KUKA KRL program: MASTER_125_LADO_B.src, MASTER_125_LADO_B.dat

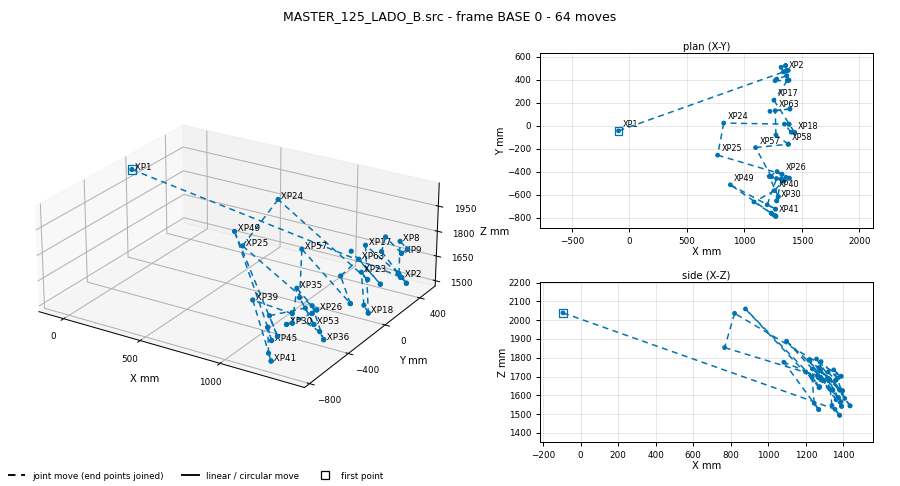
[picture p0: tool path of MASTER_125_LADO_B.src in frame BASE 0, 64 of 66 moves have a stored position in this frame; points joined in program order, loops and branches not executed]
--- MASTER_125_LADO_B.src ---
&ACCESS RVP
&REL 169
&PARAM EDITMASK = *
&PARAM TEMPLATE = C:\KRC\Roboter\Template\vorgabe
&PARAM DISKPATH = KRC:\R1\Program\Solda\MASTER_125
DEF MASTER_125_LADO_B( )
;FOLD INI;%{PE}
  ;FOLD BASISTECH INI
    GLOBAL INTERRUPT DECL 3 WHEN $STOPMESS==TRUE DO IR_STOPM ( )
    INTERRUPT ON 3
    BAS (#INITMOV,0 )
  ;ENDFOLD (BASISTECH INI)
  ;FOLD USER INI
    ;Make your modifications here

  ;ENDFOLD (USER INI)
;ENDFOLD (INI)
;FOLD OUT 128 'Perfil livre mesa B' State=FALSE CONT;%{PE}%R 8.3.48,%MKUKATPBASIS,%COUT,%VOUTX,%P 2:128, 3:Perfil livre mesa B, 5:FALSE, 6:CONTINUE
CONTINUE
$OUT[128]=FALSE
;ENDFOLD
;FOLD OUT 125 'Lado A para operador' State=TRUE ;%{PE}%R 8.3.48,%MKUKATPBASIS,%COUT,%VOUTX,%P 2:125, 3:Lado A para operador, 5:TRUE, 6:
$OUT[125]=TRUE
;ENDFOLD

;FOLD PTP HOME1 Vel=100 % PDAT2;%{PE}%R 8.3.48,%MKUKATPBASIS,%CMOVE,%VPTP,%P 1:PTP, 2:HOME1, 3:, 5:100, 7:PDAT2
$BWDSTART=FALSE
PDAT_ACT=PPDAT2
FDAT_ACT=FHOME1
BAS(#PTP_PARAMS,100)
PTP XHOME1
;ENDFOLD
;FOLD PTP P1 CONT Vel=100 % PDAT1 Tool[1]:TOCH Base[0];%{PE}%R 8.3.48,%MKUKATPBASIS,%CMOVE,%VPTP,%P 1:PTP, 2:P1, 3:C_DIS, 5:100, 7:PDAT1
$BWDSTART=FALSE
PDAT_ACT=PPDAT1
FDAT_ACT=FP1
BAS(#PTP_PARAMS,100)
PTP XP1 C_DIS
;ENDFOLD
;FOLD PTP P2 CONT Vel=100 % PDAT3 Tool[1]:TOCH Base[0];%{PE}%R 8.3.48,%MKUKATPBASIS,%CMOVE,%VPTP,%P 1:PTP, 2:P2, 3:C_DIS, 5:100, 7:PDAT3
$BWDSTART=FALSE
PDAT_ACT=PPDAT3
FDAT_ACT=FP2
BAS(#PTP_PARAMS,100)
PTP XP2 C_DIS
;ENDFOLD
;FOLD ARCON WDAT1 PTP P3 Vel=100 % PDAT4 Tool[1]:TOCH Base[0] ;%{PE}
;FOLD Parameters ;%{h}
;Params IlfProvider=kukaroboter.arctech.arconptp; Kuka.PointName=P3; Kuka.BlendingEnabled=False; Kuka.MoveDataPtpName=PDAT4; Kuka.VelocityPtp=100; Kuka.MovementParameterFieldEnabled=True; ArcTech.WdatVarName=WDAT1; ArcTech.SeamName=
;ENDFOLD
$BWDSTART = FALSE
PDAT_ACT = PPDAT4
FDAT_ACT = FP3
BAS(#PTP_PARAMS, 100.0)
TRIGGER WHEN DISTANCE = 1 DELAY = ATBg_PreDefinitionTime DO Arc_DefineStrikeParams(1, AS_WDAT1) PRIO = -1
Arc_DefineCpPattern(#OffInAdvance, WV_WDAT1, TRUE)
PTP XP3
Arc_On(1, AS_WDAT1, ATBg_StartErrSetField[1], AW_WDAT1, WV_WDAT1, ATBg_WeldErrSetField[1], #StdArcOn, " ")
Arc_DefineCpPattern(#OnInAdvance, WV_WDAT1, TRUE)
;ENDFOLD
;FOLD ARCOFF WDAT2 LIN P4 CPDAT1 Tool[1]:TOCH Base[0] ;%{PE}
;FOLD Parameters ;%{h}
;Params IlfProvider=kukaroboter.arctech.arcofflin; Kuka.PointName=P4; Kuka.BlendingEnabled=False; Kuka.MoveDataName=CPDAT1;  Kuka.MovementParameterFieldEnabled=True; ArcTech.WdatVarName=WDAT2
;ENDFOLD
$BWDSTART = FALSE
LDAT_ACT = LCPDAT1
FDAT_ACT = FP4
BAS(#CP_PARAMS, ATBg_BAS_VELDefinition)
LIN XP4
Arc_Off(1, AC_WDAT2)
;ENDFOLD
;FOLD PTP P5 CONT Vel=100 % PDAT5 Tool[1]:TOCH Base[0];%{PE}%R 8.3.48,%MKUKATPBASIS,%CMOVE,%VPTP,%P 1:PTP, 2:P5, 3:C_DIS, 5:100, 7:PDAT5
$BWDSTART=FALSE
PDAT_ACT=PPDAT5
FDAT_ACT=FP5
BAS(#PTP_PARAMS,100)
PTP XP5 C_DIS
;ENDFOLD
;FOLD PTP P8 CONT Vel=100 % PDAT8 Tool[1]:TOCH Base[0];%{PE}%R 8.3.48,%MKUKATPBASIS,%CMOVE,%VPTP,%P 1:PTP, 2:P8, 3:C_DIS, 5:100, 7:PDAT8
$BWDSTART=FALSE
PDAT_ACT=PPDAT8
FDAT_ACT=FP8
BAS(#PTP_PARAMS,100)
PTP XP8 C_DIS
;ENDFOLD
;FOLD ARCON WDAT3 PTP P6 Vel=100 % PDAT6 Tool[1]:TOCH Base[0] ;%{PE}
;FOLD Parameters ;%{h}
;Params IlfProvider=kukaroboter.arctech.arconptp; Kuka.PointName=P6; Kuka.BlendingEnabled=False; Kuka.MoveDataPtpName=PDAT6; Kuka.VelocityPtp=100; Kuka.MovementParameterFieldEnabled=True; ArcTech.WdatVarName=WDAT3; ArcTech.SeamName=
;ENDFOLD
$BWDSTART = FALSE
PDAT_ACT = PPDAT6
FDAT_ACT = FP6
BAS(#PTP_PARAMS, 100.0)
TRIGGER WHEN DISTANCE = 1 DELAY = ATBg_PreDefinitionTime DO Arc_DefineStrikeParams(1, AS_WDAT3) PRIO = -1
Arc_DefineCpPattern(#OffInAdvance, WV_WDAT3, TRUE)
PTP XP6
Arc_On(1, AS_WDAT3, ATBg_StartErrSetField[1], AW_WDAT3, WV_WDAT3, ATBg_WeldErrSetField[1], #StdArcOn, " ")
Arc_DefineCpPattern(#OnInAdvance, WV_WDAT3, TRUE)
;ENDFOLD
;FOLD ARCON WDAT4 PTP P7 Vel=100 % PDAT7 Tool[1]:TOCH Base[0] ;%{PE}
;FOLD Parameters ;%{h}
;Params IlfProvider=kukaroboter.arctech.arconptp; Kuka.PointName=P7; Kuka.BlendingEnabled=False; Kuka.MoveDataPtpName=PDAT7; Kuka.VelocityPtp=100; Kuka.MovementParameterFieldEnabled=True; ArcTech.WdatVarName=WDAT4; ArcTech.SeamName=
;ENDFOLD
$BWDSTART = FALSE
PDAT_ACT = PPDAT7
FDAT_ACT = FP7
BAS(#PTP_PARAMS, 100.0)
TRIGGER WHEN DISTANCE = 1 DELAY = ATBg_PreDefinitionTime DO Arc_DefineStrikeParams(1, AS_WDAT4) PRIO = -1
Arc_DefineCpPattern(#OffInAdvance, WV_WDAT4, TRUE)
PTP XP7
Arc_On(1, AS_WDAT4, ATBg_StartErrSetField[1], AW_WDAT4, WV_WDAT4, ATBg_WeldErrSetField[1], #StdArcOn, " ")
Arc_DefineCpPattern(#OnInAdvance, WV_WDAT4, TRUE)
;ENDFOLD
;FOLD ; CORDAO;%{PE}%R 8.3.48,%MKUKATPBASIS,%CCOMMENT,%VNORMAL,%P 2:CORDAO
;ENDFOLD
;FOLD ARCON WDAT5 PTP P9 Vel=100 % PDAT9 Tool[1]:TOCH Base[0] ;%{PE}
;FOLD Parameters ;%{h}
;Params IlfProvider=kukaroboter.arctech.arconptp; Kuka.PointName=P9; Kuka.BlendingEnabled=False; Kuka.MoveDataPtpName=PDAT9; Kuka.VelocityPtp=100; Kuka.MovementParameterFieldEnabled=True; ArcTech.WdatVarName=WDAT5; ArcTech.SeamName=
;ENDFOLD
$BWDSTART = FALSE
PDAT_ACT = PPDAT9
FDAT_ACT = FP9
BAS(#PTP_PARAMS, 100.0)
TRIGGER WHEN DISTANCE = 1 DELAY = ATBg_PreDefinitionTime DO Arc_DefineStrikeParams(1, AS_WDAT5) PRIO = -1
Arc_DefineCpPattern(#OffInAdvance, WV_WDAT5, TRUE)
PTP XP9
Arc_On(1, AS_WDAT5, ATBg_StartErrSetField[1], AW_WDAT5, WV_WDAT5, ATBg_WeldErrSetField[1], #StdArcOn, " ")
Arc_DefineCpPattern(#OnInAdvance, WV_WDAT5, TRUE)
;ENDFOLD
;FOLD ARCOFF WDAT6 LIN P10 CPDAT2 Tool[1]:TOCH Base[0] ;%{PE}
;FOLD Parameters ;%{h}
;Params IlfProvider=kukaroboter.arctech.arcofflin; Kuka.PointName=P10; Kuka.BlendingEnabled=False; Kuka.MoveDataName=CPDAT2;  Kuka.MovementParameterFieldEnabled=True; ArcTech.WdatVarName=WDAT6
;ENDFOLD
$BWDSTART = FALSE
LDAT_ACT = LCPDAT2
FDAT_ACT = FP10
BAS(#CP_PARAMS, ATBg_BAS_VELDefinition)
LIN XP10
Arc_Off(1, AC_WDAT6)
;ENDFOLD
;FOLD PTP P11 CONT Vel=100 % PDAT10 Tool[1]:TOCH Base[0];%{PE}%R 8.3.48,%MKUKATPBASIS,%CMOVE,%VPTP,%P 1:PTP, 2:P11, 3:C_DIS, 5:100, 7:PDAT10
$BWDSTART=FALSE
PDAT_ACT=PPDAT10
FDAT_ACT=FP11
BAS(#PTP_PARAMS,100)
PTP XP11 C_DIS
;ENDFOLD
;FOLD PTP P12 CONT Vel=100 % PDAT11 Tool[1]:TOCH Base[0];%{PE}%R 8.3.48,%MKUKATPBASIS,%CMOVE,%VPTP,%P 1:PTP, 2:P12, 3:C_DIS, 5:100, 7:PDAT11
$BWDSTART=FALSE
PDAT_ACT=PPDAT11
FDAT_ACT=FP12
BAS(#PTP_PARAMS,100)
PTP XP12 C_DIS
;ENDFOLD
;FOLD PTP P15 CONT Vel=100 % PDAT13 Tool[1]:TOCH Base[0];%{PE}%R 8.3.48,%MKUKATPBASIS,%CMOVE,%VPTP,%P 1:PTP, 2:P15, 3:C_DIS, 5:100, 7:PDAT13
$BWDSTART=FALSE
PDAT_ACT=PPDAT13
FDAT_ACT=FP15
BAS(#PTP_PARAMS,100)
PTP XP15 C_DIS
;ENDFOLD
;FOLD ARCON WDAT7 PTP P13 Vel=100 % PDAT12 Tool[1]:TOCH Base[0] ;%{PE}
;FOLD Parameters ;%{h}
;Params IlfProvider=kukaroboter.arctech.arconptp; Kuka.PointName=P13; Kuka.BlendingEnabled=False; Kuka.MoveDataPtpName=PDAT12; Kuka.VelocityPtp=100; Kuka.MovementParameterFieldEnabled=True; ArcTech.WdatVarName=WDAT7; ArcTech.SeamName=
;ENDFOLD
$BWDSTART = FALSE
PDAT_ACT = PPDAT12
FDAT_ACT = FP13
BAS(#PTP_PARAMS, 100.0)
TRIGGER WHEN DISTANCE = 1 DELAY = ATBg_PreDefinitionTime DO Arc_DefineStrikeParams(1, AS_WDAT7) PRIO = -1
Arc_DefineCpPattern(#OffInAdvance, WV_WDAT7, TRUE)
PTP XP13
Arc_On(1, AS_WDAT7, ATBg_StartErrSetField[1], AW_WDAT7, WV_WDAT7, ATBg_WeldErrSetField[1], #StdArcOn, " ")
Arc_DefineCpPattern(#OnInAdvance, WV_WDAT7, TRUE)
;ENDFOLD
;FOLD ARCOFF WDAT8 LIN P14 CPDAT3 Tool[1]:TOCH Base[0] ;%{PE}
;FOLD Parameters ;%{h}
;Params IlfProvider=kukaroboter.arctech.arcofflin; Kuka.PointName=P14; Kuka.BlendingEnabled=False; Kuka.MoveDataName=CPDAT3;  Kuka.MovementParameterFieldEnabled=True; ArcTech.WdatVarName=WDAT8
;ENDFOLD
$BWDSTART = FALSE
LDAT_ACT = LCPDAT3
FDAT_ACT = FP14
BAS(#CP_PARAMS, ATBg_BAS_VELDefinition)
LIN XP14
Arc_Off(1, AC_WDAT8)
;ENDFOLD
;FOLD PTP P16 CONT Vel=100 % PDAT14 Tool[1]:TOCH Base[0];%{PE}%R 8.3.48,%MKUKATPBASIS,%CMOVE,%VPTP,%P 1:PTP, 2:P16, 3:C_DIS, 5:100, 7:PDAT14
$BWDSTART=FALSE
PDAT_ACT=PPDAT14
FDAT_ACT=FP16
BAS(#PTP_PARAMS,100)
PTP XP16 C_DIS
;ENDFOLD
;FOLD PTP P17 CONT Vel=100 % PDAT15 Tool[1]:TOCH Base[0];%{PE}%R 8.3.48,%MKUKATPBASIS,%CMOVE,%VPTP,%P 1:PTP, 2:P17, 3:C_DIS, 5:100, 7:PDAT15
$BWDSTART=FALSE
PDAT_ACT=PPDAT15
FDAT_ACT=FP17
BAS(#PTP_PARAMS,100)
PTP XP17 C_DIS
;ENDFOLD
;FOLD ; CORDAO;%{PE}%R 8.3.48,%MKUKATPBASIS,%CCOMMENT,%VNORMAL,%P 2:CORDAO
;ENDFOLD
;FOLD ARCON WDAT9 PTP P18 Vel=100 % PDAT16 Tool[1]:TOCH Base[0] ;%{PE}
;FOLD Parameters ;%{h}
;Params IlfProvider=kukaroboter.arctech.arconptp; Kuka.PointName=P18; Kuka.BlendingEnabled=False; Kuka.MoveDataPtpName=PDAT16; Kuka.VelocityPtp=100; Kuka.MovementParameterFieldEnabled=True; ArcTech.WdatVarName=WDAT9; ArcTech.SeamName=
;ENDFOLD
$BWDSTART = FALSE
PDAT_ACT = PPDAT16
FDAT_ACT = FP18
BAS(#PTP_PARAMS, 100.0)
TRIGGER WHEN DISTANCE = 1 DELAY = ATBg_PreDefinitionTime DO Arc_DefineStrikeParams(1, AS_WDAT9) PRIO = -1
Arc_DefineCpPattern(#OffInAdvance, WV_WDAT9, TRUE)
PTP XP18
Arc_On(1, AS_WDAT9, ATBg_StartErrSetField[1], AW_WDAT9, WV_WDAT9, ATBg_WeldErrSetField[1], #StdArcOn, " ")
Arc_DefineCpPattern(#OnInAdvance, WV_WDAT9, TRUE)
;ENDFOLD
;FOLD ARCOFF WDAT10 LIN P19 CPDAT4 Tool[1]:TOCH Base[0] ;%{PE}
;FOLD Parameters ;%{h}
;Params IlfProvider=kukaroboter.arctech.arcofflin; Kuka.PointName=P19; Kuka.BlendingEnabled=False; Kuka.MoveDataName=CPDAT4;  Kuka.MovementParameterFieldEnabled=True; ArcTech.WdatVarName=WDAT10
;ENDFOLD
$BWDSTART = FALSE
LDAT_ACT = LCPDAT4
FDAT_ACT = FP19
BAS(#CP_PARAMS, ATBg_BAS_VELDefinition)
LIN XP19
Arc_Off(1, AC_WDAT10)
;ENDFOLD
;FOLD PTP P20 CONT Vel=100 % PDAT17 Tool[1]:TOCH Base[0];%{PE}%R 8.3.48,%MKUKATPBASIS,%CMOVE,%VPTP,%P 1:PTP, 2:P20, 3:C_DIS, 5:100, 7:PDAT17
$BWDSTART=FALSE
PDAT_ACT=PPDAT17
FDAT_ACT=FP20
BAS(#PTP_PARAMS,100)
PTP XP20 C_DIS
;ENDFOLD
;FOLD PTP P23 CONT Vel=100 % PDAT19 Tool[1]:TOCH Base[0];%{PE}%R 8.3.48,%MKUKATPBASIS,%CMOVE,%VPTP,%P 1:PTP, 2:P23, 3:C_DIS, 5:100, 7:PDAT19
$BWDSTART=FALSE
PDAT_ACT=PPDAT19
FDAT_ACT=FP23
BAS(#PTP_PARAMS,100)
PTP XP23 C_DIS
;ENDFOLD
;FOLD ; CORDAO;%{PE}%R 8.3.48,%MKUKATPBASIS,%CCOMMENT,%VNORMAL,%P 2:CORDAO
;ENDFOLD
;FOLD ARCON WDAT11 PTP P21 Vel=100 % PDAT18 Tool[1]:TOCH Base[0] ;%{PE}
;FOLD Parameters ;%{h}
;Params IlfProvider=kukaroboter.arctech.arconptp; Kuka.PointName=P21; Kuka.BlendingEnabled=False; Kuka.MoveDataPtpName=PDAT18; Kuka.VelocityPtp=100; Kuka.MovementParameterFieldEnabled=True; ArcTech.WdatVarName=WDAT11; ArcTech.SeamName=
;ENDFOLD
$BWDSTART = FALSE
PDAT_ACT = PPDAT18
FDAT_ACT = FP21
BAS(#PTP_PARAMS, 100.0)
TRIGGER WHEN DISTANCE = 1 DELAY = ATBg_PreDefinitionTime DO Arc_DefineStrikeParams(1, AS_WDAT11) PRIO = -1
Arc_DefineCpPattern(#OffInAdvance, WV_WDAT11, TRUE)
PTP XP21
Arc_On(1, AS_WDAT11, ATBg_StartErrSetField[1], AW_WDAT11, WV_WDAT11, ATBg_WeldErrSetField[1], #StdArcOn, " ")
Arc_DefineCpPattern(#OnInAdvance, WV_WDAT11, TRUE)
;ENDFOLD
;FOLD ARCOFF WDAT12 LIN P22 CPDAT5 Tool[1]:TOCH Base[0] ;%{PE}
;FOLD Parameters ;%{h}
;Params IlfProvider=kukaroboter.arctech.arcofflin; Kuka.PointName=P22; Kuka.BlendingEnabled=False; Kuka.MoveDataName=CPDAT5;  Kuka.MovementParameterFieldEnabled=True; ArcTech.WdatVarName=WDAT12
;ENDFOLD
$BWDSTART = FALSE
LDAT_ACT = LCPDAT5
FDAT_ACT = FP22
BAS(#CP_PARAMS, ATBg_BAS_VELDefinition)
LIN XP22
Arc_Off(1, AC_WDAT12)
;ENDFOLD
;FOLD PTP P24 CONT Vel=100 % PDAT20 Tool[1]:TOCH Base[0];%{PE}%R 8.3.48,%MKUKATPBASIS,%CMOVE,%VPTP,%P 1:PTP, 2:P24, 3:C_DIS, 5:100, 7:PDAT20
$BWDSTART=FALSE
PDAT_ACT=PPDAT20
FDAT_ACT=FP24
BAS(#PTP_PARAMS,100)
PTP XP24 C_DIS
;ENDFOLD
;FOLD PTP P25 CONT Vel=100 % PDAT21 Tool[1]:TOCH Base[0];%{PE}%R 8.3.48,%MKUKATPBASIS,%CMOVE,%VPTP,%P 1:PTP, 2:P25, 3:C_DIS, 5:100, 7:PDAT21
$BWDSTART=FALSE
PDAT_ACT=PPDAT21
FDAT_ACT=FP25
BAS(#PTP_PARAMS,100)
PTP XP25 C_DIS
;ENDFOLD
;FOLD ; CORDAO;%{PE}%R 8.3.48,%MKUKATPBASIS,%CCOMMENT,%VNORMAL,%P 2:CORDAO
;ENDFOLD
;FOLD ARCON WDAT13 PTP P26 Vel=100 % PDAT22 Tool[1]:TOCH Base[0] ;%{PE}
;FOLD Parameters ;%{h}
;Params IlfProvider=kukaroboter.arctech.arconptp; Kuka.PointName=P26; Kuka.BlendingEnabled=False; Kuka.MoveDataPtpName=PDAT22; Kuka.VelocityPtp=100; Kuka.MovementParameterFieldEnabled=True; ArcTech.WdatVarName=WDAT13; ArcTech.SeamName=
;ENDFOLD
$BWDSTART = FALSE
PDAT_ACT = PPDAT22
FDAT_ACT = FP26
BAS(#PTP_PARAMS, 100.0)
TRIGGER WHEN DISTANCE = 1 DELAY = ATBg_PreDefinitionTime DO Arc_DefineStrikeParams(1, AS_WDAT13) PRIO = -1
Arc_DefineCpPattern(#OffInAdvance, WV_WDAT13, TRUE)
PTP XP26
Arc_On(1, AS_WDAT13, ATBg_StartErrSetField[1], AW_WDAT13, WV_WDAT13, ATBg_WeldErrSetField[1], #StdArcOn, " ")
Arc_DefineCpPattern(#OnInAdvance, WV_WDAT13, TRUE)
;ENDFOLD
;FOLD ARCOFF WDAT14 LIN P27 CPDAT6 Tool[1]:TOCH Base[0] ;%{PE}
;FOLD Parameters ;%{h}
;Params IlfProvider=kukaroboter.arctech.arcofflin; Kuka.PointName=P27; Kuka.BlendingEnabled=False; Kuka.MoveDataName=CPDAT6;  Kuka.MovementParameterFieldEnabled=True; ArcTech.WdatVarName=WDAT14
;ENDFOLD
$BWDSTART = FALSE
LDAT_ACT = LCPDAT6
FDAT_ACT = FP27
BAS(#CP_PARAMS, ATBg_BAS_VELDefinition)
LIN XP27
Arc_Off(1, AC_WDAT14)
;ENDFOLD
;FOLD ; CORDAO;%{PE}%R 8.3.48,%MKUKATPBASIS,%CCOMMENT,%VNORMAL,%P 2:CORDAO
;ENDFOLD
;FOLD ARCON WDAT15 PTP P28 Vel=100 % PDAT23 Tool[1]:TOCH Base[0] ;%{PE}
;FOLD Parameters ;%{h}
;Params IlfProvider=kukaroboter.arctech.arconptp; Kuka.PointName=P28; Kuka.BlendingEnabled=False; Kuka.MoveDataPtpName=PDAT23; Kuka.VelocityPtp=100; Kuka.MovementParameterFieldEnabled=True; ArcTech.WdatVarName=WDAT15; ArcTech.SeamName=
;ENDFOLD
$BWDSTART = FALSE
PDAT_ACT = PPDAT23
FDAT_ACT = FP28
BAS(#PTP_PARAMS, 100.0)
TRIGGER WHEN DISTANCE = 1 DELAY = ATBg_PreDefinitionTime DO Arc_DefineStrikeParams(1, AS_WDAT15) PRIO = -1
Arc_DefineCpPattern(#OffInAdvance, WV_WDAT15, TRUE)
PTP XP28
Arc_On(1, AS_WDAT15, ATBg_StartErrSetField[1], AW_WDAT15, WV_WDAT15, ATBg_WeldErrSetField[1], #StdArcOn, " ")
Arc_DefineCpPattern(#OnInAdvance, WV_WDAT15, TRUE)
;ENDFOLD
;FOLD ARCOFF WDAT16 LIN P29 CPDAT7 Tool[1]:TOCH Base[0] ;%{PE}
;FOLD Parameters ;%{h}
;Params IlfProvider=kukaroboter.arctech.arcofflin; Kuka.PointName=P29; Kuka.BlendingEnabled=False; Kuka.MoveDataName=CPDAT7;  Kuka.MovementParameterFieldEnabled=True; ArcTech.WdatVarName=WDAT16
;ENDFOLD
$BWDSTART = FALSE
LDAT_ACT = LCPDAT7
FDAT_ACT = FP29
BAS(#CP_PARAMS, ATBg_BAS_VELDefinition)
LIN XP29
Arc_Off(1, AC_WDAT16)
;ENDFOLD
;FOLD ; CORDAO;%{PE}%R 8.3.48,%MKUKATPBASIS,%CCOMMENT,%VNORMAL,%P 2:CORDAO
;ENDFOLD
;FOLD ARCON WDAT17 PTP P30 Vel=100 % PDAT24 Tool[1]:TOCH Base[0] ;%{PE}
;FOLD Parameters ;%{h}
;Params IlfProvider=kukaroboter.arctech.arconptp; Kuka.PointName=P30; Kuka.BlendingEnabled=False; Kuka.MoveDataPtpName=PDAT24; Kuka.VelocityPtp=100; Kuka.MovementParameterFieldEnabled=True; ArcTech.WdatVarName=WDAT17; ArcTech.SeamName=
;ENDFOLD
$BWDSTART = FALSE
PDAT_ACT = PPDAT24
FDAT_ACT = FP30
BAS(#PTP_PARAMS, 100.0)
TRIGGER WHEN DISTANCE = 1 DELAY = ATBg_PreDefinitionTime DO Arc_DefineStrikeParams(1, AS_WDAT17) PRIO = -1
Arc_DefineCpPattern(#OffInAdvance, WV_WDAT17, TRUE)
PTP XP30
Arc_On(1, AS_WDAT17, ATBg_StartErrSetField[1], AW_WDAT17, WV_WDAT17, ATBg_WeldErrSetField[1], #StdArcOn, " ")
Arc_DefineCpPattern(#OnInAdvance, WV_WDAT17, TRUE)
;ENDFOLD
;FOLD ARCOFF WDAT18 LIN P31 CPDAT8 Tool[1]:TOCH Base[0] ;%{PE}
;FOLD Parameters ;%{h}
;Params IlfProvider=kukaroboter.arctech.arcofflin; Kuka.PointName=P31; Kuka.BlendingEnabled=False; Kuka.MoveDataName=CPDAT8;  Kuka.MovementParameterFieldEnabled=True; ArcTech.WdatVarName=WDAT18
;ENDFOLD
$BWDSTART = FALSE
LDAT_ACT = LCPDAT8
FDAT_ACT = FP31
BAS(#CP_PARAMS, ATBg_BAS_VELDefinition)
LIN XP31
Arc_Off(1, AC_WDAT18)
;ENDFOLD
;FOLD ; CORDAO;%{PE}%R 8.3.48,%MKUKATPBASIS,%CCOMMENT,%VNORMAL,%P 2:CORDAO
;ENDFOLD
;FOLD ARCON WDAT19 PTP P32 Vel=100 % PDAT25 Tool[1]:TOCH Base[0] ;%{PE}
;FOLD Parameters ;%{h}
;Params IlfProvider=kukaroboter.arctech.arconptp; Kuka.PointName=P32; Kuka.BlendingEnabled=False; Kuka.MoveDataPtpName=PDAT25; Kuka.VelocityPtp=100; Kuka.MovementParameterFieldEnabled=True; ArcTech.WdatVarName=WDAT19; ArcTech.SeamName=
;ENDFOLD
$BWDSTART = FALSE
PDAT_ACT = PPDAT25
FDAT_ACT = FP32
BAS(#PTP_PARAMS, 100.0)
TRIGGER WHEN DISTANCE = 1 DELAY = ATBg_PreDefinitionTime DO Arc_DefineStrikeParams(1, AS_WDAT19) PRIO = -1
Arc_DefineCpPattern(#OffInAdvance, WV_WDAT19, TRUE)
PTP XP32
Arc_On(1, AS_WDAT19, ATBg_StartErrSetField[1], AW_WDAT19, WV_WDAT19, ATBg_WeldErrSetField[1], #StdArcOn, " ")
Arc_DefineCpPattern(#OnInAdvance, WV_WDAT19, TRUE)
;ENDFOLD
;FOLD ARCOFF WDAT20 LIN P33 CPDAT9 Tool[1]:TOCH Base[0] ;%{PE}
;FOLD Parameters ;%{h}
;Params IlfProvider=kukaroboter.arctech.arcofflin; Kuka.PointName=P33; Kuka.BlendingEnabled=False; Kuka.MoveDataName=CPDAT9;  Kuka.MovementParameterFieldEnabled=True; ArcTech.WdatVarName=WDAT20
;ENDFOLD
$BWDSTART = FALSE
LDAT_ACT = LCPDAT9
FDAT_ACT = FP33
BAS(#CP_PARAMS, ATBg_BAS_VELDefinition)
LIN XP33
Arc_Off(1, AC_WDAT20)
;ENDFOLD
;FOLD PTP P35 CONT Vel=100 % PDAT27 Tool[1]:TOCH Base[0];%{PE}%R 8.3.48,%MKUKATPBASIS,%CMOVE,%VPTP,%P 1:PTP, 2:P35, 3:C_DIS, 5:100, 7:PDAT27
$BWDSTART=FALSE
PDAT_ACT=PPDAT27
FDAT_ACT=FP35
BAS(#PTP_PARAMS,100)
PTP XP35 C_DIS
;ENDFOLD
;FOLD PTP P34 CONT Vel=100 % PDAT26 Tool[1]:TOCH Base[0];%{PE}%R 8.3.48,%MKUKATPBASIS,%CMOVE,%VPTP,%P 1:PTP, 2:P34, 3:C_DIS, 5:100, 7:PDAT26
$BWDSTART=FALSE
PDAT_ACT=PPDAT26
FDAT_ACT=FP34
BAS(#PTP_PARAMS,100)
PTP XP34 C_DIS
;ENDFOLD
;FOLD ; CORDAO;%{PE}%R 8.3.48,%MKUKATPBASIS,%CCOMMENT,%VNORMAL,%P 2:CORDAO
;ENDFOLD
;FOLD ARCON WDAT21 PTP P36 Vel=100 % PDAT28 Tool[1]:TOCH Base[0] ;%{PE}
;FOLD Parameters ;%{h}
;Params IlfProvider=kukaroboter.arctech.arconptp; Kuka.PointName=P36; Kuka.BlendingEnabled=False; Kuka.MoveDataPtpName=PDAT28; Kuka.VelocityPtp=100; Kuka.MovementParameterFieldEnabled=True; ArcTech.WdatVarName=WDAT21; ArcTech.SeamName=
;ENDFOLD
$BWDSTART = FALSE
PDAT_ACT = PPDAT28
FDAT_ACT = FP36
BAS(#PTP_PARAMS, 100.0)
TRIGGER WHEN DISTANCE = 1 DELAY = ATBg_PreDefinitionTime DO Arc_DefineStrikeParams(1, AS_WDAT21) PRIO = -1
Arc_DefineCpPattern(#OffInAdvance, WV_WDAT21, TRUE)
PTP XP36
Arc_On(1, AS_WDAT21, ATBg_StartErrSetField[1], AW_WDAT21, WV_WDAT21, ATBg_WeldErrSetField[1], #StdArcOn, " ")
Arc_DefineCpPattern(#OnInAdvance, WV_WDAT21, TRUE)
;ENDFOLD
;FOLD ARCOFF WDAT22 LIN P37 CPDAT10 Tool[1]:TOCH Base[0] ;%{PE}
;FOLD Parameters ;%{h}
;Params IlfProvider=kukaroboter.arctech.arcofflin; Kuka.PointName=P37; Kuka.BlendingEnabled=False; Kuka.MoveDataName=CPDAT10;  Kuka.MovementParameterFieldEnabled=True; ArcTech.WdatVarName=WDAT22
;ENDFOLD
$BWDSTART = FALSE
LDAT_ACT = LCPDAT10
FDAT_ACT = FP37
BAS(#CP_PARAMS, ATBg_BAS_VELDefinition)
LIN XP37
Arc_Off(1, AC_WDAT22)
;ENDFOLD
;FOLD PTP P38 CONT Vel=100 % PDAT29 Tool[1]:TOCH Base[0];%{PE}%R 8.3.48,%MKUKATPBASIS,%CMOVE,%VPTP,%P 1:PTP, 2:P38, 3:C_DIS, 5:100, 7:PDAT29
$BWDSTART=FALSE
PDAT_ACT=PPDAT29
FDAT_ACT=FP38
BAS(#PTP_PARAMS,100)
PTP XP38 C_DIS
;ENDFOLD
;FOLD PTP P40 CONT Vel=100 % PDAT31 Tool[1]:TOCH Base[0];%{PE}%R 8.3.48,%MKUKATPBASIS,%CMOVE,%VPTP,%P 1:PTP, 2:P40, 3:C_DIS, 5:100, 7:PDAT31
$BWDSTART=FALSE
PDAT_ACT=PPDAT31
FDAT_ACT=FP40
BAS(#PTP_PARAMS,100)
PTP XP40 C_DIS
;ENDFOLD
;FOLD PTP P39 CONT Vel=100 % PDAT30 Tool[1]:TOCH Base[0];%{PE}%R 8.3.48,%MKUKATPBASIS,%CMOVE,%VPTP,%P 1:PTP, 2:P39, 3:C_DIS, 5:100, 7:PDAT30
$BWDSTART=FALSE
PDAT_ACT=PPDAT30
FDAT_ACT=FP39
BAS(#PTP_PARAMS,100)
PTP XP39 C_DIS
;ENDFOLD
;FOLD ; CORDAO;%{PE}%R 8.3.48,%MKUKATPBASIS,%CCOMMENT,%VNORMAL,%P 2:CORDAO
;ENDFOLD
;FOLD ARCON WDAT23 PTP P41 Vel=100 % PDAT32 Tool[1]:TOCH Base[0] ;%{PE}
;FOLD Parameters ;%{h}
;Params IlfProvider=kukaroboter.arctech.arconptp; Kuka.PointName=P41; Kuka.BlendingEnabled=False; Kuka.MoveDataPtpName=PDAT32; Kuka.VelocityPtp=100; Kuka.MovementParameterFieldEnabled=True; ArcTech.WdatVarName=WDAT23; ArcTech.SeamName=
;ENDFOLD
$BWDSTART = FALSE
PDAT_ACT = PPDAT32
FDAT_ACT = FP41
BAS(#PTP_PARAMS, 100.0)
TRIGGER WHEN DISTANCE = 1 DELAY = ATBg_PreDefinitionTime DO Arc_DefineStrikeParams(1, AS_WDAT23) PRIO = -1
Arc_DefineCpPattern(#OffInAdvance, WV_WDAT23, TRUE)
PTP XP41
Arc_On(1, AS_WDAT23, ATBg_StartErrSetField[1], AW_WDAT23, WV_WDAT23, ATBg_WeldErrSetField[1], #StdArcOn, " ")
Arc_DefineCpPattern(#OnInAdvance, WV_WDAT23, TRUE)
;ENDFOLD
;FOLD ARCOFF WDAT24 LIN P42 CPDAT11 Tool[1]:TOCH Base[0] ;%{PE}
;FOLD Parameters ;%{h}
;Params IlfProvider=kukaroboter.arctech.arcofflin; Kuka.PointName=P42; Kuka.BlendingEnabled=False; Kuka.MoveDataName=CPDAT11;  Kuka.MovementParameterFieldEnabled=True; ArcTech.WdatVarName=WDAT24
;ENDFOLD
$BWDSTART = FALSE
LDAT_ACT = LCPDAT11
FDAT_ACT = FP42
BAS(#CP_PARAMS, ATBg_BAS_VELDefinition)
LIN XP42
Arc_Off(1, AC_WDAT24)
;ENDFOLD
;FOLD PTP P43 CONT Vel=100 % PDAT33 Tool[1]:TOCH Base[0];%{PE}%R 8.3.48,%MKUKATPBASIS,%CMOVE,%VPTP,%P 1:PTP, 2:P43, 3:C_DIS, 5:100, 7:PDAT33
$BWDSTART=FALSE
PDAT_ACT=PPDAT33
FDAT_ACT=FP43
BAS(#PTP_PARAMS,100)
PTP XP43 C_DIS
;ENDFOLD
;FOLD PTP P47 CONT Vel=100 % PDAT36 Tool[1]:TOCH Base[0];%{PE}%R 8.3.48,%MKUKATPBASIS,%CMOVE,%VPTP,%P 1:PTP, 2:P47, 3:C_DIS, 5:100, 7:PDAT36
$BWDSTART=FALSE
PDAT_ACT=PPDAT36
FDAT_ACT=FP47
BAS(#PTP_PARAMS,100)
PTP XP47 C_DIS
;ENDFOLD
;FOLD ; CORDAO;%{PE}%R 8.3.48,%MKUKATPBASIS,%CCOMMENT,%VNORMAL,%P 2:CORDAO
;ENDFOLD
;FOLD ARCON WDAT25 PTP P45 Vel=100 % PDAT35 Tool[1]:TOCH Base[0] ;%{PE}
;FOLD Parameters ;%{h}
;Params IlfProvider=kukaroboter.arctech.arconptp; Kuka.PointName=P45; Kuka.BlendingEnabled=False; Kuka.MoveDataPtpName=PDAT35; Kuka.VelocityPtp=100; Kuka.MovementParameterFieldEnabled=True; ArcTech.WdatVarName=WDAT25; ArcTech.SeamName=
;ENDFOLD
$BWDSTART = FALSE
PDAT_ACT = PPDAT35
FDAT_ACT = FP45
BAS(#PTP_PARAMS, 100.0)
TRIGGER WHEN DISTANCE = 1 DELAY = ATBg_PreDefinitionTime DO Arc_DefineStrikeParams(1, AS_WDAT25) PRIO = -1
Arc_DefineCpPattern(#OffInAdvance, WV_WDAT25, TRUE)
PTP XP45
Arc_On(1, AS_WDAT25, ATBg_StartErrSetField[1], AW_WDAT25, WV_WDAT25, ATBg_WeldErrSetField[1], #StdArcOn, " ")
Arc_DefineCpPattern(#OnInAdvance, WV_WDAT25, TRUE)
;ENDFOLD
;FOLD ARCOFF WDAT26 LIN P46 CPDAT12 Tool[1]:TOCH Base[0] ;%{PE}
;FOLD Parameters ;%{h}
;Params IlfProvider=kukaroboter.arctech.arcofflin; Kuka.PointName=P46; Kuka.BlendingEnabled=False; Kuka.MoveDataName=CPDAT12;  Kuka.MovementParameterFieldEnabled=True; ArcTech.WdatVarName=WDAT26
;ENDFOLD
$BWDSTART = FALSE
LDAT_ACT = LCPDAT12
FDAT_ACT = FP46
BAS(#CP_PARAMS, ATBg_BAS_VELDefinition)
LIN XP46
Arc_Off(1, AC_WDAT26)
;ENDFOLD
;FOLD PTP P48 CONT Vel=100 % PDAT37 Tool[1]:TOCH Base[0];%{PE}%R 8.3.48,%MKUKATPBASIS,%CMOVE,%VPTP,%P 1:PTP, 2:P48, 3:C_DIS, 5:100, 7:PDAT37
$BWDSTART=FALSE
PDAT_ACT=PPDAT37
FDAT_ACT=FP48
BAS(#PTP_PARAMS,100)
PTP XP48 C_DIS
;ENDFOLD
;FOLD PTP P49 CONT Vel=100 % PDAT38 Tool[1]:TOCH Base[0];%{PE}%R 8.3.48,%MKUKATPBASIS,%CMOVE,%VPTP,%P 1:PTP, 2:P49, 3:C_DIS, 5:100, 7:PDAT38
$BWDSTART=FALSE
PDAT_ACT=PPDAT38
FDAT_ACT=FP49
BAS(#PTP_PARAMS,100)
PTP XP49 C_DIS
;ENDFOLD
;FOLD ; CORDAO;%{PE}%R 8.3.48,%MKUKATPBASIS,%CCOMMENT,%VNORMAL,%P 2:CORDAO
;ENDFOLD
;FOLD ARCON WDAT27 PTP P50 Vel=100 % PDAT39 Tool[1]:TOCH Base[0] ;%{PE}
;FOLD Parameters ;%{h}
;Params IlfProvider=kukaroboter.arctech.arconptp; Kuka.PointName=P50; Kuka.BlendingEnabled=False; Kuka.MoveDataPtpName=PDAT39; Kuka.VelocityPtp=100; Kuka.MovementParameterFieldEnabled=True; ArcTech.WdatVarName=WDAT27; ArcTech.SeamName=
;ENDFOLD
$BWDSTART = FALSE
PDAT_ACT = PPDAT39
FDAT_ACT = FP50
BAS(#PTP_PARAMS, 100.0)
TRIGGER WHEN DISTANCE = 1 DELAY = ATBg_PreDefinitionTime DO Arc_DefineStrikeParams(1, AS_WDAT27) PRIO = -1
Arc_DefineCpPattern(#OffInAdvance, WV_WDAT27, TRUE)
PTP XP50
Arc_On(1, AS_WDAT27, ATBg_StartErrSetField[1], AW_WDAT27, WV_WDAT27, ATBg_WeldErrSetField[1], #StdArcOn, " ")
Arc_DefineCpPattern(#OnInAdvance, WV_WDAT27, TRUE)
;ENDFOLD
;FOLD ARCOFF WDAT28 LIN P51 CPDAT13 Tool[1]:TOCH Base[0] ;%{PE}
;FOLD Parameters ;%{h}
;Params IlfProvider=kukaroboter.arctech.arcofflin; Kuka.PointName=P51; Kuka.BlendingEnabled=False; Kuka.MoveDataName=CPDAT13;  Kuka.MovementParameterFieldEnabled=True; ArcTech.WdatVarName=WDAT28
;ENDFOLD
$BWDSTART = FALSE
LDAT_ACT = LCPDAT13
FDAT_ACT = FP51
BAS(#CP_PARAMS, ATBg_BAS_VELDefinition)
LIN XP51
Arc_Off(1, AC_WDAT28)
;ENDFOLD
;FOLD PTP P52 CONT Vel=100 % PDAT40 Tool[1]:TOCH Base[0];%{PE}%R 8.3.48,%MKUKATPBASIS,%CMOVE,%VPTP,%P 1:PTP, 2:P52, 3:C_DIS, 5:100, 7:PDAT40
$BWDSTART=FALSE
PDAT_ACT=PPDAT40
FDAT_ACT=FP52
BAS(#PTP_PARAMS,100)
PTP XP52 C_DIS
;ENDFOLD
;FOLD PTP P55 CONT Vel=100 % PDAT42 Tool[1]:TOCH Base[0];%{PE}%R 8.3.48,%MKUKATPBASIS,%CMOVE,%VPTP,%P 1:PTP, 2:P55, 3:C_DIS, 5:100, 7:PDAT42
$BWDSTART=FALSE
PDAT_ACT=PPDAT42
FDAT_ACT=FP55
BAS(#PTP_PARAMS,100)
PTP XP55 C_DIS
;ENDFOLD
;FOLD ; CORDAO;%{PE}%R 8.3.48,%MKUKATPBASIS,%CCOMMENT,%VNORMAL,%P 2:CORDAO
;ENDFOLD
;FOLD ARCON WDAT29 PTP P53 Vel=100 % PDAT41 Tool[1]:TOCH Base[0] ;%{PE}
;FOLD Parameters ;%{h}
;Params IlfProvider=kukaroboter.arctech.arconptp; Kuka.PointName=P53; Kuka.BlendingEnabled=False; Kuka.MoveDataPtpName=PDAT41; Kuka.VelocityPtp=100; Kuka.MovementParameterFieldEnabled=True; ArcTech.WdatVarName=WDAT29; ArcTech.SeamName=
;ENDFOLD
$BWDSTART = FALSE
PDAT_ACT = PPDAT41
FDAT_ACT = FP53
BAS(#PTP_PARAMS, 100.0)
TRIGGER WHEN DISTANCE = 1 DELAY = ATBg_PreDefinitionTime DO Arc_DefineStrikeParams(1, AS_WDAT29) PRIO = -1
Arc_DefineCpPattern(#OffInAdvance, WV_WDAT29, TRUE)
PTP XP53
Arc_On(1, AS_WDAT29, ATBg_StartErrSetField[1], AW_WDAT29, WV_WDAT29, ATBg_WeldErrSetField[1], #StdArcOn, " ")
Arc_DefineCpPattern(#OnInAdvance, WV_WDAT29, TRUE)
;ENDFOLD
;FOLD ARCOFF WDAT30 LIN P54 CPDAT14 Tool[1]:TOCH Base[0] ;%{PE}
;FOLD Parameters ;%{h}
;Params IlfProvider=kukaroboter.arctech.arcofflin; Kuka.PointName=P54; Kuka.BlendingEnabled=False; Kuka.MoveDataName=CPDAT14;  Kuka.MovementParameterFieldEnabled=True; ArcTech.WdatVarName=WDAT30
;ENDFOLD
$BWDSTART = FALSE
LDAT_ACT = LCPDAT14
FDAT_ACT = FP54
BAS(#CP_PARAMS, ATBg_BAS_VELDefinition)
LIN XP54
Arc_Off(1, AC_WDAT30)
;ENDFOLD
;FOLD PTP P56 CONT Vel=100 % PDAT43 Tool[1]:TOCH Base[0];%{PE}%R 8.3.48,%MKUKATPBASIS,%CMOVE,%VPTP,%P 1:PTP, 2:P56, 3:C_DIS, 5:100, 7:PDAT43
$BWDSTART=FALSE
PDAT_ACT=PPDAT43
FDAT_ACT=FP56
BAS(#PTP_PARAMS,100)
PTP XP56 C_DIS
;ENDFOLD
;FOLD PTP P57 CONT Vel=100 % PDAT44 Tool[1]:TOCH Base[0];%{PE}%R 8.3.48,%MKUKATPBASIS,%CMOVE,%VPTP,%P 1:PTP, 2:P57, 3:C_DIS, 5:100, 7:PDAT44
$BWDSTART=FALSE
PDAT_ACT=PPDAT44
FDAT_ACT=FP57
BAS(#PTP_PARAMS,100)
PTP XP57 C_DIS
;ENDFOLD
;FOLD ; CORDAO;%{PE}%R 8.3.48,%MKUKATPBASIS,%CCOMMENT,%VNORMAL,%P 2:CORDAO
;ENDFOLD
;FOLD PTP P58 Vel=100 % PDAT45 Tool[1]:TOCH Base[0];%{PE}%R 8.3.48,%MKUKATPBASIS,%CMOVE,%VPTP,%P 1:PTP, 2:P58, 3:, 5:100, 7:PDAT45
$BWDSTART=FALSE
PDAT_ACT=PPDAT45
FDAT_ACT=FP58
BAS(#PTP_PARAMS,100)
PTP XP58
;ENDFOLD
;FOLD ARCON WDAT31 PTP P59 Vel=100 % PDAT46 Tool[1]:TOCH Base[0] ;%{PE}
;FOLD Parameters ;%{h}
;Params IlfProvider=kukaroboter.arctech.arconptp; Kuka.PointName=P59; Kuka.BlendingEnabled=False; Kuka.MoveDataPtpName=PDAT46; Kuka.VelocityPtp=100; Kuka.MovementParameterFieldEnabled=True; ArcTech.WdatVarName=WDAT31; ArcTech.SeamName=
;ENDFOLD
$BWDSTART = FALSE
PDAT_ACT = PPDAT46
FDAT_ACT = FP59
BAS(#PTP_PARAMS, 100.0)
TRIGGER WHEN DISTANCE = 1 DELAY = ATBg_PreDefinitionTime DO Arc_DefineStrikeParams(1, AS_WDAT31) PRIO = -1
Arc_DefineCpPattern(#OffInAdvance, WV_WDAT31, TRUE)
PTP XP59
Arc_On(1, AS_WDAT31, ATBg_StartErrSetField[1], AW_WDAT31, WV_WDAT31, ATBg_WeldErrSetField[1], #StdArcOn, " ")
Arc_DefineCpPattern(#OnInAdvance, WV_WDAT31, TRUE)
;ENDFOLD
;FOLD ARCOFF WDAT32 LIN P60 CPDAT15 Tool[1]:TOCH Base[0] ;%{PE}
;FOLD Parameters ;%{h}
;Params IlfProvider=kukaroboter.arctech.arcofflin; Kuka.PointName=P60; Kuka.BlendingEnabled=False; Kuka.MoveDataName=CPDAT15;  Kuka.MovementParameterFieldEnabled=True; ArcTech.WdatVarName=WDAT32
;ENDFOLD
$BWDSTART = FALSE
LDAT_ACT = LCPDAT15
FDAT_ACT = FP60
BAS(#CP_PARAMS, ATBg_BAS_VELDefinition)
LIN XP60
Arc_Off(1, AC_WDAT32)
;ENDFOLD
;FOLD PTP P64 Vel=100 % PDAT49 Tool[1]:TOCH Base[0];%{PE}%R 8.3.48,%MKUKATPBASIS,%CMOVE,%VPTP,%P 1:PTP, 2:P64, 3:, 5:100, 7:PDAT49
$BWDSTART=FALSE
PDAT_ACT=PPDAT49
FDAT_ACT=FP64
BAS(#PTP_PARAMS,100)
PTP XP64
;ENDFOLD
;FOLD PTP P63 Vel=100 % PDAT48 Tool[1]:TOCH Base[0];%{PE}%R 8.3.48,%MKUKATPBASIS,%CMOVE,%VPTP,%P 1:PTP, 2:P63, 3:, 5:100, 7:PDAT48
$BWDSTART=FALSE
PDAT_ACT=PPDAT48
FDAT_ACT=FP63
BAS(#PTP_PARAMS,100)
PTP XP63
;ENDFOLD
;FOLD ; CORDAO;%{PE}%R 8.3.48,%MKUKATPBASIS,%CCOMMENT,%VNORMAL,%P 2:CORDAO
;ENDFOLD
;FOLD ARCON WDAT33 PTP P61 Vel=100 % PDAT47 Tool[1]:TOCH Base[0] ;%{PE}
;FOLD Parameters ;%{h}
;Params IlfProvider=kukaroboter.arctech.arconptp; Kuka.PointName=P61; Kuka.BlendingEnabled=False; Kuka.MoveDataPtpName=PDAT47; Kuka.VelocityPtp=100; Kuka.MovementParameterFieldEnabled=True; ArcTech.WdatVarName=WDAT33; ArcTech.SeamName=
;ENDFOLD
$BWDSTART = FALSE
PDAT_ACT = PPDAT47
FDAT_ACT = FP61
BAS(#PTP_PARAMS, 100.0)
TRIGGER WHEN DISTANCE = 1 DELAY = ATBg_PreDefinitionTime DO Arc_DefineStrikeParams(1, AS_WDAT33) PRIO = -1
Arc_DefineCpPattern(#OffInAdvance, WV_WDAT33, TRUE)
PTP XP61
Arc_On(1, AS_WDAT33, ATBg_StartErrSetField[1], AW_WDAT33, WV_WDAT33, ATBg_WeldErrSetField[1], #StdArcOn, " ")
Arc_DefineCpPattern(#OnInAdvance, WV_WDAT33, TRUE)
;ENDFOLD
;FOLD ARCOFF WDAT34 LIN P62 CPDAT16 Tool[1]:TOCH Base[0] ;%{PE}
;FOLD Parameters ;%{h}
;Params IlfProvider=kukaroboter.arctech.arcofflin; Kuka.PointName=P62; Kuka.BlendingEnabled=False; Kuka.MoveDataName=CPDAT16;  Kuka.MovementParameterFieldEnabled=True; ArcTech.WdatVarName=WDAT34
;ENDFOLD
$BWDSTART = FALSE
LDAT_ACT = LCPDAT16
FDAT_ACT = FP62
BAS(#CP_PARAMS, ATBg_BAS_VELDefinition)
LIN XP62
Arc_Off(1, AC_WDAT34)
;ENDFOLD
;FOLD PTP P65 Vel=100 % PDAT50 Tool[1]:TOCH Base[0];%{PE}%R 8.3.48,%MKUKATPBASIS,%CMOVE,%VPTP,%P 1:PTP, 2:P65, 3:, 5:100, 7:PDAT50
$BWDSTART=FALSE
PDAT_ACT=PPDAT50
FDAT_ACT=FP65
BAS(#PTP_PARAMS,100)
PTP XP65
;ENDFOLD
;FOLD PTP home1 Vel=100 % PDAT51;%{PE}%R 8.3.48,%MKUKATPBASIS,%CMOVE,%VPTP,%P 1:PTP, 2:home1, 3:, 5:100, 7:PDAT51
$BWDSTART=FALSE
PDAT_ACT=PPDAT51
FDAT_ACT=Fhome1
BAS(#PTP_PARAMS,100)
PTP Xhome1
;ENDFOLD
;FOLD WAIT FOR NOT ( IN 128 'AVA/REC MESA A' );%{PE}%R 8.3.48,%MKUKATPBASIS,%CEXT_WAIT_FOR,%VEXT_WAIT_FOR,%P 2:NOT, 4:, 5:$IN, 6:128, 7:AVA/REC MESA A, 9:
WAIT FOR  NOT ( $IN[128] )
;ENDFOLD
END

--- MASTER_125_LADO_B.dat ---
&ACCESS RVP
&REL 169
&PARAM EDITMASK = *
&PARAM TEMPLATE = C:\KRC\Roboter\Template\vorgabe
&PARAM DISKPATH = KRC:\R1\Program\Solda\MASTER_125
DEFDAT  MASTER_125_LADO_B
;FOLD EXTERNAL DECLARATIONS;%{PE}%MKUKATPBASIS,%CEXT,%VCOMMON,%P
;FOLD BASISTECH EXT;%{PE}%MKUKATPBASIS,%CEXT,%VEXT,%P
EXT  BAS (BAS_COMMAND  :IN,REAL  :IN )
DECL INT SUCCESS
;ENDFOLD (BASISTECH EXT)
;FOLD USER EXT;%{E}%MKUKATPUSER,%CEXT,%VEXT,%P
;Make your modifications here

;ENDFOLD (USER EXT)
;ENDFOLD (EXTERNAL DECLARATIONS)
DECL BASIS_SUGG_T LAST_BASIS={POINT1[] "P65                     ",POINT2[] "P65                     ",CP_PARAMS[] "CPDAT0                  ",PTP_PARAMS[] "PDAT51                  ",CONT[] "                        ",CP_VEL[] "2.0                     ",PTP_VEL[] "100                     ",SYNC_PARAMS[] "SYNCDAT                 ",SPL_NAME[] "S0                      ",A_PARAMS[] "ADAT0                   "}
DECL E6POS XP1={X -93.6792068,Y -45.7907486,Z 2038.98669,A 6.74064255,B 69.8344269,C 88.5610428,S 3,T 11,E1 15.0002480,E2 15.0049477,E3 14.9978313,E4 0.0,E5 0.0,E6 0.0}
DECL FDAT FP1={TOOL_NO 1,BASE_NO 0,IPO_FRAME #BASE,POINT2[] " ",TQ_STATE FALSE}
DECL PDAT PPDAT1={VEL 100.000,ACC 30.0000,APO_DIST 100.000,APO_MODE #CDIS,GEAR_JERK 50.0000,EXAX_IGN 3}
DECL FDAT Fhome1={TOOL_NO 1,BASE_NO 0,IPO_FRAME #BASE,POINT2[] " ",TQ_STATE FALSE}
DECL PDAT PPDAT2={VEL 100.000,ACC 100.000,APO_DIST 100.000,GEAR_JERK 50.0000,EXAX_IGN 3}
DECL E6POS XP2={X 1355.22070,Y 471.588196,Z 1525.90491,A 152.644531,B 59.4338760,C -132.086304,S 0,T 43,E1 15.0002480,E2 15.0049477,E3 14.9978313,E4 0.0,E5 0.0,E6 0.0}
DECL FDAT FP2={TOOL_NO 1,BASE_NO 0,IPO_FRAME #BASE,POINT2[] " ",TQ_STATE FALSE}
DECL PDAT PPDAT3={VEL 100.000,ACC 100.000,APO_DIST 100.000,APO_MODE #CDIS,GEAR_JERK 50.0000,EXAX_IGN 3}
DECL ATBg_Start_T AS_WDAT1={JobModeId -187662529,ParamSetId 687014726,StartTime 0.0,PreFlowTime 0.100000,Channel1 30.0000,Channel2 1.00000,Channel3 0.0,Channel4 0.0,Channel5 0.0,Channel6 0.0,Channel7 0.0,Channel8 0.0,PurgeTime 0.0}
DECL ATBg_Weld_T AW_WDAT1={JobModeId -187662529,ParamSetId -430485013,Velocity 0.00830000,Channel1 30.0000,Channel2 1.00000,Channel3 0.0,Channel4 0.0,Channel5 0.0,Channel6 0.0,Channel7 0.0,Channel8 0.0}
DECL WTCg_WeaveDefinition_T WV_WDAT1={Pattern #None,Length 4.00000,Amplitude 2.00000,Angle 0.0}
DECL FDAT FP3={TOOL_NO 1,BASE_NO 0,IPO_FRAME #BASE,POINT2[] " ",TQ_STATE FALSE}
DECL PDAT PPDAT4={ACC 100.000,APO_DIST 100.000,APO_MODE #CPTP,GEAR_JERK 50.0000}
DECL E6POS XP3={X 1380.06152,Y 480.134125,Z 1493.73,A 154.326157,B 58.4383507,C -130.123260,S 0,T 43,E1 15.0002480,E2 15.0049477,E3 14.9978313,E4 0.0,E5 0.0,E6 0.0}
DECL MODULEPARAM_T LAST_TP_PARAMS={PARAMS[] "Kuka.MoveDataPtpName=PDAT47; Kuka.VelocityPtp=100; Kuka.PointName=P62; Kuka.BlendingEnabled=False; Kuka.FrameData.tq_state=False; Kuka.FrameData.base_no=0; Kuka.FrameData.tool_no=1; Kuka.FrameData.ipo_frame=#BASE; Kuka.MovementDataPdat.apo_mode=#CPTP; Kuka.MovementDataPdat.apo_dist=100; Kuka.MovementData.acc=100; Kuka.MovementData.gear_jerk=50; ArcTech.WdatVarName=WDAT34; Kuka.MoveDataName=CPDAT16; Kuka.VelocityPath=2; Kuka.MovementData.apo_fac=50; Kuka.MovementData.apo_dist=100; Kuka.MovementData.axis_acc=100; Kuka.MovementData.axis_vel=100; Kuka.MovementData.circ_typ=#BASE; Kuka.MovementData.exax_ign=0; Kuka.MovementData.jerk_fac=50; Kuka.MovementData.ori_typ=#VAR                                                              "}
DECL ATBg_Crater_T AC_WDAT2={JobModeId -187662529,ParamSetId -1375177600,CraterTime 0.100000,PostflowTime 0.100000,Channel1 30.0000,Channel2 1.00000,Channel3 0.0,Channel4 0.0,Channel5 0.0,Channel6 0.0,Channel7 0.0,Channel8 0.0,BurnBackTime 0.0}
DECL FDAT FP4={TOOL_NO 1,BASE_NO 0,IPO_FRAME #BASE,POINT2[] " ",TQ_STATE FALSE}
DECL LDAT LCPDAT1={ACC 100.000,APO_DIST 100.000,APO_FAC 50.0000,AXIS_VEL 100.000,AXIS_ACC 100.000,ORI_TYP #VAR,CIRC_TYP #BASE,JERK_FAC 50.0000,GEAR_JERK 50.0000,EXAX_IGN 0}
DECL E6POS XP4={X 1380.06152,Y 480.134125,Z 1493.73,A 154.326157,B 58.4383507,C -130.123260,S 0,T 43,E1 15.0002480,E2 15.0049477,E3 14.9978313,E4 0.0,E5 0.0,E6 0.0}
DECL E6POS XP5={X 1339.25940,Y 466.097076,Z 1545.74817,A 151.529938,B 60.0425072,C -133.376709,S 0,T 43,E1 15.0002480,E2 15.0049477,E3 14.9978313,E4 0.0,E5 0.0,E6 0.0}
DECL FDAT FP5={TOOL_NO 1,BASE_NO 0,IPO_FRAME #BASE,POINT2[] " ",TQ_STATE FALSE}
DECL PDAT PPDAT5={VEL 100.000,ACC 100.000,APO_DIST 100.000,APO_MODE #CDIS,GEAR_JERK 50.0000,EXAX_IGN 3}
DECL ATBg_Start_T AS_WDAT3={JobModeId -187662529,ParamSetId 687014726,StartTime 0.0,PreFlowTime 0.100000,Channel1 30.0000,Channel2 1.00000,Channel3 0.0,Channel4 0.0,Channel5 0.0,Channel6 0.0,Channel7 0.0,Channel8 0.0,PurgeTime 0.0}
DECL ATBg_Weld_T AW_WDAT3={JobModeId -187662529,ParamSetId -430485013,Velocity 0.00830000,Channel1 30.0000,Channel2 1.00000,Channel3 0.0,Channel4 0.0,Channel5 0.0,Channel6 0.0,Channel7 0.0,Channel8 0.0}
DECL WTCg_WeaveDefinition_T WV_WDAT3={Pattern #None,Length 4.00000,Amplitude 2.00000,Angle 0.0}
DECL FDAT FP6={TOOL_NO 1,BASE_NO 0,IPO_FRAME #BASE,POINT2[] " ",TQ_STATE FALSE}
DECL PDAT PPDAT6={ACC 100.000,APO_DIST 100.000,APO_MODE #CPTP,GEAR_JERK 50.0000}
DECL E6POS XP6={X 1358.82751,Y 521.879272,Z 1679.82361,A -17.4242783,B -53.8819923,C -57.1328506,S 2,T 11,E1 15.0002480,E2 15.0049477,E3 14.9978313,E4 0.0,E5 0.0,E6 0.0}
DECL ATBg_Start_T AS_WDAT4={JobModeId -187662529,ParamSetId 687014726,StartTime 0.0,PreFlowTime 0.100000,Channel1 30.0000,Channel2 1.00000,Channel3 0.0,Channel4 0.0,Channel5 0.0,Channel6 0.0,Channel7 0.0,Channel8 0.0,PurgeTime 0.0}
DECL ATBg_Weld_T AW_WDAT4={JobModeId -187662529,ParamSetId -430485013,Velocity 0.00830000,Channel1 30.0000,Channel2 1.00000,Channel3 0.0,Channel4 0.0,Channel5 0.0,Channel6 0.0,Channel7 0.0,Channel8 0.0}
DECL WTCg_WeaveDefinition_T WV_WDAT4={Pattern #None,Length 4.00000,Amplitude 2.00000,Angle 0.0}
DECL FDAT FP7={TOOL_NO 1,BASE_NO 0,IPO_FRAME #BASE,POINT2[] " ",TQ_STATE FALSE}
DECL PDAT PPDAT7={ACC 100.000,APO_DIST 100.000,APO_MODE #CPTP,GEAR_JERK 50.0000}
DECL E6POS XP7={X 1358.82751,Y 521.879272,Z 1679.82361,A -17.4242783,B -53.8819923,C -57.1328506,S 2,T 11,E1 15.0002480,E2 15.0049477,E3 14.9978313,E4 0.0,E5 0.0,E6 0.0}
DECL E6POS XP8={X 1318.95911,Y 506.413696,Z 1723.69519,A -19.1788177,B -55.3923492,C -54.9816399,S 2,T 11,E1 15.0002480,E2 15.0049477,E3 14.9978313,E4 0.0,E5 0.0,E6 0.0}
DECL FDAT FP8={TOOL_NO 1,BASE_NO 0,IPO_FRAME #BASE,POINT2[] " ",TQ_STATE FALSE}
DECL PDAT PPDAT8={VEL 100.000,ACC 100.000,APO_DIST 100.000,APO_MODE #CDIS,GEAR_JERK 50.0000,EXAX_IGN 3}
DECL ATBg_Start_T AS_WDAT5={JobModeId -187662529,ParamSetId 687014726,StartTime 0.0,PreFlowTime 0.100000,Channel1 30.0000,Channel2 1.00000,Channel3 0.0,Channel4 0.0,Channel5 0.0,Channel6 0.0,Channel7 0.0,Channel8 0.0,PurgeTime 0.0}
DECL ATBg_Weld_T AW_WDAT5={JobModeId -187662529,ParamSetId -430485013,Velocity 0.00830000,Channel1 30.0000,Channel2 1.00000,Channel3 0.0,Channel4 0.0,Channel5 0.0,Channel6 0.0,Channel7 0.0,Channel8 0.0}
DECL WTCg_WeaveDefinition_T WV_WDAT5={Pattern #None,Length 4.00000,Amplitude 2.00000,Angle 0.0}
DECL FDAT FP9={TOOL_NO 1,BASE_NO 0,IPO_FRAME #BASE,POINT2[] " ",TQ_STATE FALSE}
DECL PDAT PPDAT9={ACC 100.000,APO_DIST 100.000,APO_MODE #CPTP,GEAR_JERK 50.0000}
DECL E6POS XP9={X 1368.33142,Y 432.711487,Z 1691.14160,A -28.8243904,B -51.5982552,C -49.9969673,S 2,T 11,E1 15.0002480,E2 15.0049477,E3 14.9978313,E4 0.0,E5 0.0,E6 0.0}
DECL ATBg_Crater_T AC_WDAT6={JobModeId -187662529,ParamSetId -1375177600,CraterTime 0.100000,PostflowTime 0.100000,Channel1 30.0000,Channel2 1.00000,Channel3 0.0,Channel4 0.0,Channel5 0.0,Channel6 0.0,Channel7 0.0,Channel8 0.0,BurnBackTime 0.0}
DECL FDAT FP10={TOOL_NO 1,BASE_NO 0,IPO_FRAME #BASE,POINT2[] " ",TQ_STATE FALSE}
DECL LDAT LCPDAT2={ACC 100.000,APO_DIST 100.000,APO_FAC 50.0000,AXIS_VEL 100.000,AXIS_ACC 100.000,ORI_TYP #VAR,CIRC_TYP #BASE,JERK_FAC 50.0000,GEAR_JERK 50.0000,EXAX_IGN 0}
DECL E6POS XP10={X 1368.33142,Y 432.711487,Z 1691.14160,A -28.8243904,B -51.5982552,C -49.9969673,S 2,T 11,E1 15.0002480,E2 15.0049477,E3 14.9978313,E4 0.0,E5 0.0,E6 0.0}
DECL E6POS XP11={X 1281.30579,Y 404.254,Z 1779.42419,A -32.9022102,B -54.2787933,C -44.8894730,S 2,T 11,E1 15.0002480,E2 15.0049477,E3 14.9978313,E4 0.0,E5 0.0,E6 0.0}
DECL FDAT FP11={TOOL_NO 1,BASE_NO 0,IPO_FRAME #BASE,POINT2[] " ",TQ_STATE FALSE}
DECL PDAT PPDAT10={VEL 100.000,ACC 100.000,APO_DIST 100.000,APO_MODE #CDIS,GEAR_JERK 50.0000,EXAX_IGN 3}
DECL E6POS XP12={X 1266.71875,Y 390.163666,Z 1693.92737,A 99.9351807,B 84.8981094,C 171.781036,S 2,T 43,E1 15.0002480,E2 15.0049477,E3 14.9978313,E4 0.0,E5 0.0,E6 0.0}
DECL FDAT FP12={TOOL_NO 1,BASE_NO 0,IPO_FRAME #BASE,POINT2[] " ",TQ_STATE FALSE}
DECL PDAT PPDAT11={VEL 100.000,ACC 100.000,APO_DIST 100.000,APO_MODE #CDIS,GEAR_JERK 50.0000,EXAX_IGN 3}
DECL ATBg_Start_T AS_WDAT7={JobModeId -187662529,ParamSetId 687014726,StartTime 0.0,PreFlowTime 0.100000,Channel1 30.0000,Channel2 1.00000,Channel3 0.0,Channel4 0.0,Channel5 0.0,Channel6 0.0,Channel7 0.0,Channel8 0.0,PurgeTime 0.0}
DECL ATBg_Weld_T AW_WDAT7={JobModeId -187662529,ParamSetId -430485013,Velocity 0.00830000,Channel1 30.0000,Channel2 1.00000,Channel3 0.0,Channel4 0.0,Channel5 0.0,Channel6 0.0,Channel7 0.0,Channel8 0.0}
DECL WTCg_WeaveDefinition_T WV_WDAT7={Pattern #None,Length 4.00000,Amplitude 2.00000,Angle 0.0}
DECL FDAT FP13={TOOL_NO 1,BASE_NO 0,IPO_FRAME #BASE,POINT2[] " ",TQ_STATE FALSE}
DECL PDAT PPDAT12={ACC 100.000,APO_DIST 100.000,APO_MODE #CPTP,GEAR_JERK 50.0000}
DECL E6POS XP13={X 1386.53833,Y 394.780365,Z 1565.15125,A 114.637604,B 66.0098419,C -154.524185,S 2,T 35,E1 15.0002480,E2 15.0049477,E3 14.9978313,E4 0.0,E5 0.0,E6 0.0}
DECL ATBg_Crater_T AC_WDAT8={JobModeId -187662529,ParamSetId -1375177600,CraterTime 0.100000,PostflowTime 0.100000,Channel1 30.0000,Channel2 1.00000,Channel3 0.0,Channel4 0.0,Channel5 0.0,Channel6 0.0,Channel7 0.0,Channel8 0.0,BurnBackTime 0.0}
DECL FDAT FP14={TOOL_NO 1,BASE_NO 0,IPO_FRAME #BASE,POINT2[] " ",TQ_STATE FALSE}
DECL LDAT LCPDAT3={ACC 100.000,APO_DIST 100.000,APO_FAC 50.0000,AXIS_VEL 100.000,AXIS_ACC 100.000,ORI_TYP #VAR,CIRC_TYP #BASE,JERK_FAC 50.0000,GEAR_JERK 50.0000,EXAX_IGN 0}
DECL E6POS XP14={X 1386.53833,Y 394.780365,Z 1565.15125,A 114.637604,B 66.0098419,C -154.524185,S 2,T 35,E1 15.0002480,E2 15.0049477,E3 14.9978313,E4 0.0,E5 0.0,E6 0.0}
DECL E6POS XP15={X 1373.60938,Y 391.658539,Z 1587.77356,A 112.168297,B 66.5700150,C -157.855301,S 2,T 35,E1 15.0002480,E2 15.0049477,E3 14.9978313,E4 0.0,E5 0.0,E6 0.0}
DECL FDAT FP15={TOOL_NO 1,BASE_NO 0,IPO_FRAME #BASE,POINT2[] " ",TQ_STATE FALSE}
DECL PDAT PPDAT13={VEL 100.000,ACC 100.000,APO_DIST 100.000,APO_MODE #CDIS,GEAR_JERK 50.0000,EXAX_IGN 3}
DECL E6POS XP16={X 1373.60938,Y 391.658539,Z 1587.77356,A 112.168297,B 66.5700150,C -157.855301,S 2,T 35,E1 15.0002480,E2 15.0049477,E3 14.9978313,E4 0.0,E5 0.0,E6 0.0}
DECL FDAT FP16={TOOL_NO 1,BASE_NO 0,IPO_FRAME #BASE,POINT2[] " ",TQ_STATE FALSE}
DECL PDAT PPDAT14={VEL 100.000,ACC 100.000,APO_DIST 100.000,APO_MODE #CDIS,GEAR_JERK 50.0000,EXAX_IGN 3}
DECL E6POS XP17={X 1257.02148,Y 220.533508,Z 1793.28052,A 73.7259521,B 63.1257324,C 166.202835,S 0,T 35,E1 15.0002480,E2 15.0049477,E3 14.9978313,E4 0.0,E5 0.0,E6 0.0}
DECL FDAT FP17={TOOL_NO 1,BASE_NO 0,IPO_FRAME #BASE,POINT2[] " ",TQ_STATE FALSE}
DECL PDAT PPDAT15={VEL 100.000,ACC 100.000,APO_DIST 100.000,APO_MODE #CDIS,GEAR_JERK 50.0000,EXAX_IGN 3}
DECL ATBg_Start_T AS_WDAT9={JobModeId -187662529,ParamSetId 687014726,StartTime 0.0,PreFlowTime 0.100000,Channel1 30.0000,Channel2 1.00000,Channel3 0.0,Channel4 0.0,Channel5 0.0,Channel6 0.0,Channel7 0.0,Channel8 0.0,PurgeTime 0.0}
DECL ATBg_Weld_T AW_WDAT9={JobModeId -187662529,ParamSetId -430485013,Velocity 0.00830000,Channel1 30.0000,Channel2 1.00000,Channel3 0.0,Channel4 0.0,Channel5 0.0,Channel6 0.0,Channel7 0.0,Channel8 0.0}
DECL WTCg_WeaveDefinition_T WV_WDAT9={Pattern #None,Length 4.00000,Amplitude 2.00000,Angle 0.0}
DECL FDAT FP18={TOOL_NO 1,BASE_NO 0,IPO_FRAME #BASE,POINT2[] " ",TQ_STATE FALSE}
DECL PDAT PPDAT16={ACC 100.000,APO_DIST 100.000,APO_MODE #CPTP,GEAR_JERK 50.0000}
DECL E6POS XP18={X 1435.53638,Y -58.7056313,Z 1543.86975,A 175.892319,B 73.4190216,C -92.0082474,S 2,T 34,E1 15.0002480,E2 15.0049477,E3 14.9978313,E4 0.0,E5 0.0,E6 0.0}
DECL ATBg_Crater_T AC_WDAT10={JobModeId -187662529,ParamSetId -1375177600,CraterTime 0.100000,PostflowTime 0.100000,Channel1 30.0000,Channel2 1.00000,Channel3 0.0,Channel4 0.0,Channel5 0.0,Channel6 0.0,Channel7 0.0,Channel8 0.0,BurnBackTime 0.0}
DECL FDAT FP19={TOOL_NO 1,BASE_NO 0,IPO_FRAME #BASE,POINT2[] " ",TQ_STATE FALSE}
DECL LDAT LCPDAT4={ACC 100.000,APO_DIST 100.000,APO_FAC 50.0000,AXIS_VEL 100.000,AXIS_ACC 100.000,ORI_TYP #VAR,CIRC_TYP #BASE,JERK_FAC 50.0000,GEAR_JERK 50.0000,EXAX_IGN 0}
DECL E6POS XP19={X 1435.53638,Y -58.7056313,Z 1543.86975,A 175.892319,B 73.4190216,C -92.0082474,S 2,T 34,E1 15.0002480,E2 15.0049477,E3 14.9978313,E4 0.0,E5 0.0,E6 0.0}
DECL E6POS XP20={X 1407.46729,Y -58.2145309,Z 1583.13550,A 175.429581,B 75.6171722,C -92.4883194,S 2,T 34,E1 15.0002480,E2 15.0049477,E3 14.9978313,E4 0.0,E5 0.0,E6 0.0}
DECL FDAT FP20={TOOL_NO 1,BASE_NO 0,IPO_FRAME #BASE,POINT2[] " ",TQ_STATE FALSE}
DECL PDAT PPDAT17={VEL 100.000,ACC 100.000,APO_DIST 100.000,APO_MODE #CDIS,GEAR_JERK 50.0000,EXAX_IGN 3}
DECL ATBg_Start_T AS_WDAT11={JobModeId -187662529,ParamSetId 687014726,StartTime 0.0,PreFlowTime 0.100000,Channel1 30.0000,Channel2 1.00000,Channel3 0.0,Channel4 0.0,Channel5 0.0,Channel6 0.0,Channel7 0.0,Channel8 0.0,PurgeTime 0.0}
DECL ATBg_Weld_T AW_WDAT11={JobModeId -187662529,ParamSetId -430485013,Velocity 0.00830000,Channel1 30.0000,Channel2 1.00000,Channel3 0.0,Channel4 0.0,Channel5 0.0,Channel6 0.0,Channel7 0.0,Channel8 0.0}
DECL WTCg_WeaveDefinition_T WV_WDAT11={Pattern #None,Length 4.00000,Amplitude 2.00000,Angle 0.0}
DECL FDAT FP21={TOOL_NO 1,BASE_NO 0,IPO_FRAME #BASE,POINT2[] " ",TQ_STATE FALSE}
DECL PDAT PPDAT18={ACC 100.000,APO_DIST 100.000,APO_MODE #CPTP,GEAR_JERK 50.0000}
DECL E6POS XP21={X 1387.86279,Y 11.8383608,Z 1701.27014,A 13.2442245,B -66.8493881,C -104.105347,S 2,T 2,E1 15.0002480,E2 15.0049477,E3 14.9978313,E4 0.0,E5 0.0,E6 0.0}
DECL ATBg_Crater_T AC_WDAT12={JobModeId -187662529,ParamSetId -1375177600,CraterTime 0.100000,PostflowTime 0.100000,Channel1 30.0000,Channel2 1.00000,Channel3 0.0,Channel4 0.0,Channel5 0.0,Channel6 0.0,Channel7 0.0,Channel8 0.0,BurnBackTime 0.0}
DECL FDAT FP22={TOOL_NO 1,BASE_NO 0,IPO_FRAME #BASE,POINT2[] " ",TQ_STATE FALSE}
DECL LDAT LCPDAT5={ACC 100.000,APO_DIST 100.000,APO_FAC 50.0000,AXIS_VEL 100.000,AXIS_ACC 100.000,ORI_TYP #VAR,CIRC_TYP #BASE,JERK_FAC 50.0000,GEAR_JERK 50.0000,EXAX_IGN 0}
DECL E6POS XP22={X 1387.86279,Y 11.8383608,Z 1701.27014,A 13.2442245,B -66.8493881,C -104.105347,S 2,T 2,E1 15.0002480,E2 15.0049477,E3 14.9978313,E4 0.0,E5 0.0,E6 0.0}
DECL E6POS XP23={X 1348.58960,Y 12.5254889,Z 1735.26257,A 14.1632328,B -68.2945786,C -105.099472,S 2,T 2,E1 15.0002480,E2 15.0049477,E3 14.9978313,E4 0.0,E5 0.0,E6 0.0}
DECL FDAT FP23={TOOL_NO 1,BASE_NO 0,IPO_FRAME #BASE,POINT2[] " ",TQ_STATE FALSE}
DECL PDAT PPDAT19={VEL 100.000,ACC 100.000,APO_DIST 100.000,APO_MODE #CDIS,GEAR_JERK 50.0000,EXAX_IGN 3}
DECL E6POS XP24={X 820.690125,Y 21.7616539,Z 2036.55139,A 58.3905487,B -83.5455246,C -150.197540,S 2,T 2,E1 15.0002480,E2 15.0049477,E3 14.9978313,E4 0.0,E5 0.0,E6 0.0}
DECL FDAT FP24={TOOL_NO 1,BASE_NO 0,IPO_FRAME #BASE,POINT2[] " ",TQ_STATE FALSE}
DECL PDAT PPDAT20={VEL 100.000,ACC 100.000,APO_DIST 100.000,APO_MODE #CDIS,GEAR_JERK 50.0000,EXAX_IGN 3}
DECL E6POS XP25={X 767.516113,Y -257.017578,Z 1854.10425,A 115.753975,B 85.3225555,C -136.753128,S 2,T 34,E1 15.0002480,E2 15.0049477,E3 14.9978313,E4 0.0,E5 0.0,E6 0.0}
DECL FDAT FP25={TOOL_NO 1,BASE_NO 0,IPO_FRAME #BASE,POINT2[] " ",TQ_STATE FALSE}
DECL PDAT PPDAT21={VEL 100.000,ACC 100.000,APO_DIST 100.000,APO_MODE #CDIS,GEAR_JERK 50.0000,EXAX_IGN 3}
DECL ATBg_Start_T AS_WDAT13={JobModeId -187662529,ParamSetId 687014726,StartTime 0.0,PreFlowTime 0.100000,Channel1 30.0000,Channel2 1.00000,Channel3 0.0,Channel4 0.0,Channel5 0.0,Channel6 0.0,Channel7 0.0,Channel8 0.0,PurgeTime 0.0}
DECL ATBg_Weld_T AW_WDAT13={JobModeId -187662529,ParamSetId -430485013,Velocity 0.00830000,Channel1 30.0000,Channel2 1.00000,Channel3 0.0,Channel4 0.0,Channel5 0.0,Channel6 0.0,Channel7 0.0,Channel8 0.0}
DECL WTCg_WeaveDefinition_T WV_WDAT13={Pattern #None,Length 4.00000,Amplitude 2.00000,Angle 0.0}
DECL FDAT FP26={TOOL_NO 1,BASE_NO 0,IPO_FRAME #BASE,POINT2[] " ",TQ_STATE FALSE}
DECL PDAT PPDAT22={ACC 100.000,APO_DIST 100.000,APO_MODE #CPTP,GEAR_JERK 50.0000}
DECL E6POS XP26={X 1326.43164,Y -422.607,Z 1682.74353,A -15.4735899,B 66.0405579,C 90.7537537,S 6,T 50,E1 15.0002480,E2 15.0049477,E3 14.9978313,E4 0.0,E5 0.0,E6 0.0}
DECL ATBg_Crater_T AC_WDAT14={JobModeId -187662529,ParamSetId -1375177600,CraterTime 0.100000,PostflowTime 0.100000,Channel1 30.0000,Channel2 1.00000,Channel3 0.0,Channel4 0.0,Channel5 0.0,Channel6 0.0,Channel7 0.0,Channel8 0.0,BurnBackTime 0.0}
DECL FDAT FP27={TOOL_NO 1,BASE_NO 0,IPO_FRAME #BASE,POINT2[] " ",TQ_STATE FALSE}
DECL LDAT LCPDAT6={ACC 100.000,APO_DIST 100.000,APO_FAC 50.0000,AXIS_VEL 100.000,AXIS_ACC 100.000,ORI_TYP #VAR,CIRC_TYP #BASE,JERK_FAC 50.0000,GEAR_JERK 50.0000,EXAX_IGN 0}
DECL E6POS XP27={X 1326.43164,Y -422.607,Z 1682.74353,A -15.4735899,B 66.0405579,C 90.7537537,S 6,T 50,E1 15.0002480,E2 15.0049477,E3 14.9978313,E4 0.0,E5 0.0,E6 0.0}
DECL ATBg_Start_T AS_WDAT15={JobModeId -187662529,ParamSetId 687014726,StartTime 0.0,PreFlowTime 0.100000,Channel1 30.0000,Channel2 1.00000,Channel3 0.0,Channel4 0.0,Channel5 0.0,Channel6 0.0,Channel7 0.0,Channel8 0.0,PurgeTime 0.0}
DECL ATBg_Weld_T AW_WDAT15={JobModeId -187662529,ParamSetId -430485013,Velocity 0.00830000,Channel1 30.0000,Channel2 1.00000,Channel3 0.0,Channel4 0.0,Channel5 0.0,Channel6 0.0,Channel7 0.0,Channel8 0.0}
DECL WTCg_WeaveDefinition_T WV_WDAT15={Pattern #None,Length 4.00000,Amplitude 2.00000,Angle 0.0}
DECL FDAT FP28={TOOL_NO 1,BASE_NO 0,IPO_FRAME #BASE,POINT2[] " ",TQ_STATE FALSE}
DECL PDAT PPDAT23={ACC 100.000,APO_DIST 100.000,APO_MODE #CPTP,GEAR_JERK 50.0000}
DECL E6POS XP28={X 1321.95422,Y -463.511780,Z 1678.22131,A -26.0240803,B 66.0559464,C 81.9989319,S 6,T 50,E1 15.0002480,E2 15.0049477,E3 14.9978313,E4 0.0,E5 0.0,E6 0.0}
DECL ATBg_Crater_T AC_WDAT16={JobModeId -187662529,ParamSetId -1375177600,CraterTime 0.100000,PostflowTime 0.100000,Channel1 30.0000,Channel2 1.00000,Channel3 0.0,Channel4 0.0,Channel5 0.0,Channel6 0.0,Channel7 0.0,Channel8 0.0,BurnBackTime 0.0}
DECL FDAT FP29={TOOL_NO 1,BASE_NO 0,IPO_FRAME #BASE,POINT2[] " ",TQ_STATE FALSE}
DECL LDAT LCPDAT7={ACC 100.000,APO_DIST 100.000,APO_FAC 50.0000,AXIS_VEL 100.000,AXIS_ACC 100.000,ORI_TYP #VAR,CIRC_TYP #BASE,JERK_FAC 50.0000,GEAR_JERK 50.0000,EXAX_IGN 0}
DECL E6POS XP29={X 1321.95422,Y -463.511780,Z 1678.22131,A -26.0240803,B 66.0559464,C 81.9989319,S 6,T 50,E1 15.0002480,E2 15.0049477,E3 14.9978313,E4 0.0,E5 0.0,E6 0.0}
DECL ATBg_Start_T AS_WDAT17={JobModeId -187662529,ParamSetId 687014726,StartTime 0.0,PreFlowTime 0.100000,Channel1 30.0000,Channel2 1.00000,Channel3 0.0,Channel4 0.0,Channel5 0.0,Channel6 0.0,Channel7 0.0,Channel8 0.0,PurgeTime 0.0}
DECL ATBg_Weld_T AW_WDAT17={JobModeId -187662529,ParamSetId -430485013,Velocity 0.00830000,Channel1 30.0000,Channel2 1.00000,Channel3 0.0,Channel4 0.0,Channel5 0.0,Channel6 0.0,Channel7 0.0,Channel8 0.0}
DECL WTCg_WeaveDefinition_T WV_WDAT17={Pattern #None,Length 4.00000,Amplitude 2.00000,Angle 0.0}
DECL FDAT FP30={TOOL_NO 1,BASE_NO 0,IPO_FRAME #BASE,POINT2[] " ",TQ_STATE FALSE}
DECL PDAT PPDAT24={ACC 100.000,APO_DIST 100.000,APO_MODE #CPTP,GEAR_JERK 50.0000}
DECL E6POS XP30={X 1281.17664,Y -653.828064,Z 1682.58142,A -43.5542641,B 67.9440842,C 72.2446136,S 6,T 50,E1 15.0002480,E2 15.0049477,E3 14.9978313,E4 0.0,E5 0.0,E6 0.0}
DECL ATBg_Crater_T AC_WDAT18={JobModeId -187662529,ParamSetId -1375177600,CraterTime 0.100000,PostflowTime 0.100000,Channel1 30.0000,Channel2 1.00000,Channel3 0.0,Channel4 0.0,Channel5 0.0,Channel6 0.0,Channel7 0.0,Channel8 0.0,BurnBackTime 0.0}
DECL FDAT FP31={TOOL_NO 1,BASE_NO 0,IPO_FRAME #BASE,POINT2[] " ",TQ_STATE FALSE}
DECL LDAT LCPDAT8={ACC 100.000,APO_DIST 100.000,APO_FAC 50.0000,AXIS_VEL 100.000,AXIS_ACC 100.000,ORI_TYP #VAR,CIRC_TYP #BASE,JERK_FAC 50.0000,GEAR_JERK 50.0000,EXAX_IGN 0}
DECL E6POS XP31={X 1281.17664,Y -653.828064,Z 1682.58142,A -43.5542641,B 67.9440842,C 72.2446136,S 6,T 50,E1 15.0002480,E2 15.0049477,E3 14.9978313,E4 0.0,E5 0.0,E6 0.0}
DECL ATBg_Start_T AS_WDAT19={JobModeId -187662529,ParamSetId 687014726,StartTime 0.0,PreFlowTime 0.100000,Channel1 30.0000,Channel2 1.00000,Channel3 0.0,Channel4 0.0,Channel5 0.0,Channel6 0.0,Channel7 0.0,Channel8 0.0,PurgeTime 0.0}
DECL ATBg_Weld_T AW_WDAT19={JobModeId -187662529,ParamSetId -430485013,Velocity 0.00830000,Channel1 30.0000,Channel2 1.00000,Channel3 0.0,Channel4 0.0,Channel5 0.0,Channel6 0.0,Channel7 0.0,Channel8 0.0}
DECL WTCg_WeaveDefinition_T WV_WDAT19={Pattern #None,Length 4.00000,Amplitude 2.00000,Angle 0.0}
DECL FDAT FP32={TOOL_NO 1,BASE_NO 0,IPO_FRAME #BASE,POINT2[] " ",TQ_STATE FALSE}
DECL PDAT PPDAT25={ACC 100.000,APO_DIST 100.000,APO_MODE #CPTP,GEAR_JERK 50.0000}
DECL E6POS XP32={X 1294.15637,Y -617.494141,Z 1678.27393,A -43.4271355,B 67.8758621,C 71.6963806,S 6,T 50,E1 15.0001621,E2 15.0047283,E3 14.9978209,E4 0.0,E5 0.0,E6 0.0}
DECL ATBg_Crater_T AC_WDAT20={JobModeId -187662529,ParamSetId -1375177600,CraterTime 0.100000,PostflowTime 0.100000,Channel1 30.0000,Channel2 1.00000,Channel3 0.0,Channel4 0.0,Channel5 0.0,Channel6 0.0,Channel7 0.0,Channel8 0.0,BurnBackTime 0.0}
DECL FDAT FP33={TOOL_NO 1,BASE_NO 0,IPO_FRAME #BASE,POINT2[] " ",TQ_STATE FALSE}
DECL LDAT LCPDAT9={ACC 100.000,APO_DIST 100.000,APO_FAC 50.0000,AXIS_VEL 100.000,AXIS_ACC 100.000,ORI_TYP #VAR,CIRC_TYP #BASE,JERK_FAC 50.0000,GEAR_JERK 50.0000,EXAX_IGN 0}
DECL E6POS XP33={X 1294.15637,Y -617.494141,Z 1678.27393,A -43.4271355,B 67.8758621,C 71.6963806,S 6,T 50,E1 15.0001621,E2 15.0047283,E3 14.9978209,E4 0.0,E5 0.0,E6 0.0}
DECL E6POS XP34={X 1284.84546,Y -399.930237,Z 1687.45605,A -142.093460,B 76.3748703,C -37.6935120,S 0,T 10,E1 15.0001621,E2 15.0047283,E3 14.9978209,E4 0.0,E5 0.0,E6 0.0}
DECL FDAT FP34={TOOL_NO 1,BASE_NO 0,IPO_FRAME #BASE,POINT2[] " ",TQ_STATE FALSE}
DECL PDAT PPDAT26={VEL 100.000,ACC 100.000,APO_DIST 100.000,APO_MODE #CDIS,GEAR_JERK 50.0000,EXAX_IGN 3}
DECL E6POS XP35={X 1215.86926,Y -441.629883,Z 1787.60925,A -48.2706070,B 77.1183929,C 69.3370132,S 2,T 34,E1 15.0001621,E2 15.0047283,E3 14.9978209,E4 0.0,E5 0.0,E6 0.0}
DECL FDAT FP35={TOOL_NO 1,BASE_NO 0,IPO_FRAME #BASE,POINT2[] " ",TQ_STATE FALSE}
DECL PDAT PPDAT27={VEL 100.000,ACC 100.000,APO_DIST 100.000,APO_MODE #CDIS,GEAR_JERK 50.0000,EXAX_IGN 3}
DECL ATBg_Start_T AS_WDAT21={JobModeId -187662529,ParamSetId 687014726,StartTime 0.0,PreFlowTime 0.100000,Channel1 30.0000,Channel2 1.00000,Channel3 0.0,Channel4 0.0,Channel5 0.0,Channel6 0.0,Channel7 0.0,Channel8 0.0,PurgeTime 0.0}
DECL ATBg_Weld_T AW_WDAT21={JobModeId -187662529,ParamSetId -430485013,Velocity 0.00830000,Channel1 30.0000,Channel2 1.00000,Channel3 0.0,Channel4 0.0,Channel5 0.0,Channel6 0.0,Channel7 0.0,Channel8 0.0}
DECL WTCg_WeaveDefinition_T WV_WDAT21={Pattern #None,Length 4.00000,Amplitude 2.00000,Angle 0.0}
DECL FDAT FP36={TOOL_NO 1,BASE_NO 0,IPO_FRAME #BASE,POINT2[] " ",TQ_STATE FALSE}
DECL PDAT PPDAT28={ACC 100.000,APO_DIST 100.000,APO_MODE #CPTP,GEAR_JERK 50.0000}
DECL E6POS XP36={X 1390.59229,Y -457.253967,Z 1541.18945,A -144.849106,B 60.2874870,C -43.2236137,S 2,T 10,E1 15.0001621,E2 15.0047283,E3 14.9978209,E4 0.0,E5 0.0,E6 0.0}
DECL ATBg_Crater_T AC_WDAT22={JobModeId -187662529,ParamSetId -1375177600,CraterTime 0.100000,PostflowTime 0.100000,Channel1 30.0000,Channel2 1.00000,Channel3 0.0,Channel4 0.0,Channel5 0.0,Channel6 0.0,Channel7 0.0,Channel8 0.0,BurnBackTime 0.0}
DECL FDAT FP37={TOOL_NO 1,BASE_NO 0,IPO_FRAME #BASE,POINT2[] " ",TQ_STATE FALSE}
DECL LDAT LCPDAT10={ACC 100.000,APO_DIST 100.000,APO_FAC 50.0000,AXIS_VEL 100.000,AXIS_ACC 100.000,ORI_TYP #VAR,CIRC_TYP #BASE,JERK_FAC 50.0000,GEAR_JERK 50.0000,EXAX_IGN 0}
DECL E6POS XP37={X 1390.59229,Y -457.253967,Z 1541.18945,A -144.849106,B 60.2874870,C -43.2236137,S 2,T 10,E1 15.0001621,E2 15.0047283,E3 14.9978209,E4 0.0,E5 0.0,E6 0.0}
DECL E6POS XP38={X 1361.23035,Y -449.002,Z 1576.86365,A -142.631,B 61.2586632,C -40.6821251,S 2,T 10,E1 15.0001621,E2 15.0047283,E3 14.9978209,E4 0.0,E5 0.0,E6 0.0}
DECL FDAT FP38={TOOL_NO 1,BASE_NO 0,IPO_FRAME #BASE,POINT2[] " ",TQ_STATE FALSE}
DECL PDAT PPDAT29={VEL 100.000,ACC 100.000,APO_DIST 100.000,APO_MODE #CDIS,GEAR_JERK 50.0000,EXAX_IGN 3}
DECL E6POS XP39={X 1082.93372,Y -663.827087,Z 1776.15735,A -112.605759,B 71.6189117,C 6.77819109,S 0,T 6,E1 15.0001621,E2 15.0047283,E3 14.9978209,E4 0.0,E5 0.0,E6 0.0}
DECL FDAT FP39={TOOL_NO 1,BASE_NO 0,IPO_FRAME #BASE,POINT2[] " ",TQ_STATE FALSE}
DECL PDAT PPDAT30={VEL 100.000,ACC 100.000,APO_DIST 100.000,APO_MODE #CDIS,GEAR_JERK 50.0000,EXAX_IGN 3}
DECL E6POS XP40={X 1262.73743,Y -565.255127,Z 1703.14514,A -116.386597,B 69.2440567,C -5.11696911,S 0,T 2,E1 15.0001621,E2 15.0047283,E3 14.9978209,E4 0.0,E5 0.0,E6 0.0}
DECL FDAT FP40={TOOL_NO 1,BASE_NO 0,IPO_FRAME #BASE,POINT2[] " ",TQ_STATE FALSE}
DECL PDAT PPDAT31={VEL 100.000,ACC 100.000,APO_DIST 100.000,APO_MODE #CDIS,GEAR_JERK 50.0000,EXAX_IGN 3}
DECL ATBg_Start_T AS_WDAT23={JobModeId -187662529,ParamSetId 687014726,StartTime 0.0,PreFlowTime 0.100000,Channel1 30.0000,Channel2 1.00000,Channel3 0.0,Channel4 0.0,Channel5 0.0,Channel6 0.0,Channel7 0.0,Channel8 0.0,PurgeTime 0.0}
DECL ATBg_Weld_T AW_WDAT23={JobModeId -187662529,ParamSetId -430485013,Velocity 0.00830000,Channel1 30.0000,Channel2 1.00000,Channel3 0.0,Channel4 0.0,Channel5 0.0,Channel6 0.0,Channel7 0.0,Channel8 0.0}
DECL WTCg_WeaveDefinition_T WV_WDAT23={Pattern #None,Length 4.00000,Amplitude 2.00000,Angle 0.0}
DECL FDAT FP41={TOOL_NO 1,BASE_NO 0,IPO_FRAME #BASE,POINT2[] " ",TQ_STATE FALSE}
DECL PDAT PPDAT32={ACC 100.000,APO_DIST 100.000,APO_MODE #CPTP,GEAR_JERK 50.0000}
DECL E6POS XP41={X 1268.46021,Y -783.802917,Z 1524.27478,A -148.481644,B 54.0366821,C -34.7950096,S 0,T 2,E1 15.0001621,E2 15.0047283,E3 14.9978209,E4 0.0,E5 0.0,E6 0.0}
DECL ATBg_Crater_T AC_WDAT24={JobModeId -187662529,ParamSetId -1375177600,CraterTime 0.100000,PostflowTime 0.100000,Channel1 30.0000,Channel2 1.00000,Channel3 0.0,Channel4 0.0,Channel5 0.0,Channel6 0.0,Channel7 0.0,Channel8 0.0,BurnBackTime 0.0}
DECL FDAT FP42={TOOL_NO 1,BASE_NO 0,IPO_FRAME #BASE,POINT2[] " ",TQ_STATE FALSE}
DECL LDAT LCPDAT11={ACC 100.000,APO_DIST 100.000,APO_FAC 50.0000,AXIS_VEL 100.000,AXIS_ACC 100.000,ORI_TYP #VAR,CIRC_TYP #BASE,JERK_FAC 50.0000,GEAR_JERK 50.0000,EXAX_IGN 0}
DECL E6POS XP42={X 1268.46021,Y -783.802917,Z 1524.27478,A -148.481644,B 54.0366821,C -34.7950096,S 0,T 2,E1 15.0001621,E2 15.0047283,E3 14.9978209,E4 0.0,E5 0.0,E6 0.0}
DECL E6POS XP43={X 1244.70093,Y -770.725220,Z 1557.23560,A -146.738831,B 54.7226448,C -32.6511650,S 0,T 2,E1 15.0001621,E2 15.0047283,E3 14.9978209,E4 0.0,E5 0.0,E6 0.0}
DECL FDAT FP43={TOOL_NO 1,BASE_NO 0,IPO_FRAME #BASE,POINT2[] " ",TQ_STATE FALSE}
DECL PDAT PPDAT33={VEL 100.000,ACC 100.000,APO_DIST 100.000,APO_MODE #CDIS,GEAR_JERK 50.0000,EXAX_IGN 3}
DECL E6POS XP44={X 1273.29175,Y -788.863708,Z 1645.08582,A 25.2739086,B -46.8869743,C -142.069244,S 2,T 34,E1 15.0001621,E2 15.0047283,E3 14.9978209,E4 0.0,E5 0.0,E6 0.0}
DECL FDAT FP44={TOOL_NO 1,BASE_NO 0,IPO_FRAME #BASE,POINT2[] " ",TQ_STATE FALSE}
DECL PDAT PPDAT34={VEL 100.000,ACC 100.000,APO_DIST 100.000,GEAR_JERK 50.0000,EXAX_IGN 3}
DECL ATBg_Start_T AS_WDAT25={JobModeId -187662529,ParamSetId 687014726,StartTime 0.0,PreFlowTime 0.100000,Channel1 30.0000,Channel2 1.00000,Channel3 0.0,Channel4 0.0,Channel5 0.0,Channel6 0.0,Channel7 0.0,Channel8 0.0,PurgeTime 0.0}
DECL ATBg_Weld_T AW_WDAT25={JobModeId -187662529,ParamSetId -430485013,Velocity 0.00830000,Channel1 30.0000,Channel2 1.00000,Channel3 0.0,Channel4 0.0,Channel5 0.0,Channel6 0.0,Channel7 0.0,Channel8 0.0}
DECL WTCg_WeaveDefinition_T WV_WDAT25={Pattern #None,Length 4.00000,Amplitude 2.00000,Angle 0.0}
DECL FDAT FP45={TOOL_NO 1,BASE_NO 0,IPO_FRAME #BASE,POINT2[] " ",TQ_STATE FALSE}
DECL PDAT PPDAT35={ACC 100.000,APO_DIST 100.000,APO_MODE #CPTP,GEAR_JERK 50.0000}
DECL E6POS XP45={X 1273.29175,Y -788.863708,Z 1645.08582,A 25.2739086,B -46.8869743,C -142.069244,S 2,T 34,E1 15.0001621,E2 15.0047283,E3 14.9978209,E4 0.0,E5 0.0,E6 0.0}
DECL ATBg_Crater_T AC_WDAT26={JobModeId -187662529,ParamSetId -1375177600,CraterTime 0.100000,PostflowTime 0.100000,Channel1 30.0000,Channel2 1.00000,Channel3 0.0,Channel4 0.0,Channel5 0.0,Channel6 0.0,Channel7 0.0,Channel8 0.0,BurnBackTime 0.0}
DECL FDAT FP46={TOOL_NO 1,BASE_NO 0,IPO_FRAME #BASE,POINT2[] " ",TQ_STATE FALSE}
DECL LDAT LCPDAT12={ACC 100.000,APO_DIST 100.000,APO_FAC 50.0000,AXIS_VEL 100.000,AXIS_ACC 100.000,ORI_TYP #VAR,CIRC_TYP #BASE,JERK_FAC 50.0000,GEAR_JERK 50.0000,EXAX_IGN 0}
DECL E6POS XP46={X 1273.29175,Y -788.863708,Z 1645.08582,A 25.2739086,B -46.8869743,C -142.069244,S 2,T 34,E1 15.0001621,E2 15.0047283,E3 14.9978209,E4 0.0,E5 0.0,E6 0.0}
DECL E6POS XP47={X 1233.19543,Y -761.008850,Z 1697.90356,A 27.4576588,B -47.9926567,C -145.034500,S 2,T 34,E1 15.0001278,E2 15.0046473,E3 14.9978094,E4 0.0,E5 0.0,E6 0.0}
DECL FDAT FP47={TOOL_NO 1,BASE_NO 0,IPO_FRAME #BASE,POINT2[] " ",TQ_STATE FALSE}
DECL PDAT PPDAT36={VEL 100.000,ACC 100.000,APO_DIST 100.000,APO_MODE #CDIS,GEAR_JERK 50.0000,EXAX_IGN 3}
DECL E6POS XP48={X 1233.19543,Y -761.008850,Z 1697.90356,A 27.4576588,B -47.9926567,C -145.034500,S 2,T 34,E1 15.0001278,E2 15.0046473,E3 14.9978094,E4 0.0,E5 0.0,E6 0.0}
DECL FDAT FP48={TOOL_NO 1,BASE_NO 0,IPO_FRAME #BASE,POINT2[] " ",TQ_STATE FALSE}
DECL PDAT PPDAT37={VEL 100.000,ACC 100.000,APO_DIST 100.000,APO_MODE #CDIS,GEAR_JERK 50.0000,EXAX_IGN 3}
DECL E6POS XP49={X 878.360413,Y -514.474792,Z 2060.12305,A 59.3534737,B -53.5727196,C 174.517410,S 0,T 34,E1 15.0001278,E2 -116.368507,E3 14.9978094,E4 0.0,E5 0.0,E6 0.0}
DECL FDAT FP49={TOOL_NO 1,BASE_NO 0,IPO_FRAME #BASE,POINT2[] " ",TQ_STATE FALSE}
DECL PDAT PPDAT38={VEL 100.000,ACC 100.000,APO_DIST 100.000,APO_MODE #CDIS,GEAR_JERK 50.0000,EXAX_IGN 3}
DECL ATBg_Start_T AS_WDAT27={JobModeId -187662529,ParamSetId 687014726,StartTime 0.0,PreFlowTime 0.100000,Channel1 30.0000,Channel2 1.00000,Channel3 0.0,Channel4 0.0,Channel5 0.0,Channel6 0.0,Channel7 0.0,Channel8 0.0,PurgeTime 0.0}
DECL ATBg_Weld_T AW_WDAT27={JobModeId -187662529,ParamSetId -430485013,Velocity 0.00830000,Channel1 30.0000,Channel2 1.00000,Channel3 0.0,Channel4 0.0,Channel5 0.0,Channel6 0.0,Channel7 0.0,Channel8 0.0}
DECL WTCg_WeaveDefinition_T WV_WDAT27={Pattern #None,Length 4.00000,Amplitude 2.00000,Angle 0.0}
DECL FDAT FP50={TOOL_NO 1,BASE_NO 0,IPO_FRAME #BASE,POINT2[] " ",TQ_STATE FALSE}
DECL PDAT PPDAT39={ACC 100.000,APO_DIST 100.000,APO_MODE #CPTP,GEAR_JERK 50.0000}
DECL E6POS XP50={X 1270.85657,Y -725.972229,Z 1641.43237,A -107.259491,B 72.6566925,C 9.48652172,S 2,T 10,E1 15.0001278,E2 -131.762726,E3 14.9978094,E4 0.0,E5 0.0,E6 0.0}
DECL ATBg_Crater_T AC_WDAT28={JobModeId -187662529,ParamSetId -1375177600,CraterTime 0.100000,PostflowTime 0.100000,Channel1 30.0000,Channel2 1.00000,Channel3 0.0,Channel4 0.0,Channel5 0.0,Channel6 0.0,Channel7 0.0,Channel8 0.0,BurnBackTime 0.0}
DECL FDAT FP51={TOOL_NO 1,BASE_NO 0,IPO_FRAME #BASE,POINT2[] " ",TQ_STATE FALSE}
DECL LDAT LCPDAT13={ACC 100.000,APO_DIST 100.000,APO_FAC 50.0000,AXIS_VEL 100.000,AXIS_ACC 100.000,ORI_TYP #VAR,CIRC_TYP #BASE,JERK_FAC 50.0000,GEAR_JERK 50.0000,EXAX_IGN 0}
DECL E6POS XP51={X 1270.85657,Y -725.972229,Z 1641.43237,A -107.259491,B 72.6566925,C 9.48652172,S 2,T 10,E1 15.0001278,E2 -131.762726,E3 14.9978094,E4 0.0,E5 0.0,E6 0.0}
DECL E6POS XP52={X 1198.73730,Y -688.058411,Z 1725.45447,A -95.9645844,B 71.6007843,C 21.3495655,S 2,T 10,E1 15.0001278,E2 -131.762726,E3 14.9978094,E4 0.0,E5 0.0,E6 0.0}
DECL FDAT FP52={TOOL_NO 1,BASE_NO 0,IPO_FRAME #BASE,POINT2[] " ",TQ_STATE FALSE}
DECL PDAT PPDAT40={VEL 100.000,ACC 100.000,APO_DIST 100.000,APO_MODE #CDIS,GEAR_JERK 50.0000,EXAX_IGN 3}
DECL ATBg_Start_T AS_WDAT29={JobModeId -187662529,ParamSetId 687014726,StartTime 0.0,PreFlowTime 0.100000,Channel1 30.0000,Channel2 1.00000,Channel3 0.0,Channel4 0.0,Channel5 0.0,Channel6 0.0,Channel7 0.0,Channel8 0.0,PurgeTime 0.0}
DECL ATBg_Weld_T AW_WDAT29={JobModeId -187662529,ParamSetId -430485013,Velocity 0.00830000,Channel1 30.0000,Channel2 1.00000,Channel3 0.0,Channel4 0.0,Channel5 0.0,Channel6 0.0,Channel7 0.0,Channel8 0.0}
DECL WTCg_WeaveDefinition_T WV_WDAT29={Pattern #None,Length 4.00000,Amplitude 2.00000,Angle 0.0}
DECL FDAT FP53={TOOL_NO 1,BASE_NO 0,IPO_FRAME #BASE,POINT2[] " ",TQ_STATE FALSE}
DECL PDAT PPDAT41={ACC 100.000,APO_DIST 100.000,APO_MODE #CPTP,GEAR_JERK 50.0000}
DECL E6POS XP53={X 1343.85339,Y -481.292603,Z 1627.28271,A -105.402840,B 81.4318237,C 1.34640944,S 2,T 10,E1 15.0001278,E2 -131.762726,E3 14.9978094,E4 0.0,E5 0.0,E6 0.0}
DECL ATBg_Crater_T AC_WDAT30={JobModeId -187662529,ParamSetId -1375177600,CraterTime 0.100000,PostflowTime 0.100000,Channel1 30.0000,Channel2 1.00000,Channel3 0.0,Channel4 0.0,Channel5 0.0,Channel6 0.0,Channel7 0.0,Channel8 0.0,BurnBackTime 0.0}
DECL FDAT FP54={TOOL_NO 1,BASE_NO 0,IPO_FRAME #BASE,POINT2[] " ",TQ_STATE FALSE}
DECL LDAT LCPDAT14={ACC 100.000,APO_DIST 100.000,APO_FAC 50.0000,AXIS_VEL 100.000,AXIS_ACC 100.000,ORI_TYP #VAR,CIRC_TYP #BASE,JERK_FAC 50.0000,GEAR_JERK 50.0000,EXAX_IGN 0}
DECL E6POS XP54={X 1343.85339,Y -481.292603,Z 1627.28271,A -105.402840,B 81.4318237,C 1.34640944,S 2,T 10,E1 15.0001278,E2 -131.762726,E3 14.9978094,E4 0.0,E5 0.0,E6 0.0}
DECL E6POS XP55={X 1279.25659,Y -460.126892,Z 1696.98523,A -85.3543,B 80.7109756,C 21.6353989,S 2,T 10,E1 15.0001278,E2 -131.762726,E3 14.9978094,E4 0.0,E5 0.0,E6 0.0}
DECL FDAT FP55={TOOL_NO 1,BASE_NO 0,IPO_FRAME #BASE,POINT2[] " ",TQ_STATE FALSE}
DECL PDAT PPDAT42={VEL 100.000,ACC 100.000,APO_DIST 100.000,APO_MODE #CDIS,GEAR_JERK 50.0000,EXAX_IGN 3}
DECL E6POS XP56={X 1235.26160,Y -445.711548,Z 1740.25867,A -74.6470413,B 79.7205048,C 32.4993591,S 2,T 10,E1 15.0001278,E2 -131.762726,E3 14.9978094,E4 0.0,E5 0.0,E6 0.0}
DECL FDAT FP56={TOOL_NO 1,BASE_NO 0,IPO_FRAME #BASE,POINT2[] " ",TQ_STATE FALSE}
DECL PDAT PPDAT43={VEL 100.000,ACC 100.000,APO_DIST 100.000,APO_MODE #CDIS,GEAR_JERK 50.0000,EXAX_IGN 3}
DECL E6POS XP57={X 1097.36914,Y -191.412735,Z 1887.94983,A -40.9607201,B 74.1731,C 56.5119438,S 2,T 10,E1 15.0001278,E2 -131.762726,E3 14.9978094,E4 0.0,E5 0.0,E6 0.0}
DECL FDAT FP57={TOOL_NO 1,BASE_NO 0,IPO_FRAME #BASE,POINT2[] " ",TQ_STATE FALSE}
DECL PDAT PPDAT44={VEL 100.000,ACC 100.000,APO_DIST 100.000,APO_MODE #CDIS,GEAR_JERK 50.0000,EXAX_IGN 3}
DECL E6POS XP58={X 1381.33386,Y -161.537140,Z 1628.13171,A -99.9627075,B 81.4212494,C -6.35471535,S 2,T 10,E1 15.0001278,E2 -131.762726,E3 14.9978094,E4 0.0,E5 0.0,E6 0.0}
DECL FDAT FP58={TOOL_NO 1,BASE_NO 0,IPO_FRAME #BASE,POINT2[] " ",TQ_STATE FALSE}
DECL PDAT PPDAT45={VEL 100.000,ACC 100.000,APO_DIST 100.000,GEAR_JERK 50.0000,EXAX_IGN 3}
DECL ATBg_Start_T AS_WDAT31={JobModeId -187662529,ParamSetId 687014726,StartTime 0.0,PreFlowTime 0.100000,Channel1 30.0000,Channel2 1.00000,Channel3 0.0,Channel4 0.0,Channel5 0.0,Channel6 0.0,Channel7 0.0,Channel8 0.0,PurgeTime 0.0}
DECL ATBg_Weld_T AW_WDAT31={JobModeId -187662529,ParamSetId -430485013,Velocity 0.00830000,Channel1 30.0000,Channel2 1.00000,Channel3 0.0,Channel4 0.0,Channel5 0.0,Channel6 0.0,Channel7 0.0,Channel8 0.0}
DECL WTCg_WeaveDefinition_T WV_WDAT31={Pattern #None,Length 4.00000,Amplitude 2.00000,Angle 0.0}
DECL FDAT FP59={TOOL_NO 1,BASE_NO 0,IPO_FRAME #BASE,POINT2[] " ",TQ_STATE FALSE}
DECL PDAT PPDAT46={ACC 100.000,APO_DIST 100.000,APO_MODE #CPTP,GEAR_JERK 50.0000}
DECL E6POS XP59={X 1381.33386,Y -161.537140,Z 1628.13171,A -99.9627075,B 81.4212494,C -6.35471535,S 2,T 10,E1 15.0001278,E2 -131.762726,E3 14.9978094,E4 0.0,E5 0.0,E6 0.0}
DECL ATBg_Crater_T AC_WDAT32={JobModeId -187662529,ParamSetId -1375177600,CraterTime 0.100000,PostflowTime 0.100000,Channel1 30.0000,Channel2 1.00000,Channel3 0.0,Channel4 0.0,Channel5 0.0,Channel6 0.0,Channel7 0.0,Channel8 0.0,BurnBackTime 0.0}
DECL FDAT FP60={TOOL_NO 1,BASE_NO 0,IPO_FRAME #BASE,POINT2[] " ",TQ_STATE FALSE}
DECL LDAT LCPDAT15={ACC 100.000,APO_DIST 100.000,APO_FAC 50.0000,AXIS_VEL 100.000,AXIS_ACC 100.000,ORI_TYP #VAR,CIRC_TYP #BASE,JERK_FAC 50.0000,GEAR_JERK 50.0000,EXAX_IGN 0}
DECL E6POS XP60={X 1381.33386,Y -161.537140,Z 1628.13171,A -99.9627075,B 81.4212494,C -6.35471535,S 2,T 10,E1 15.0001278,E2 -131.762726,E3 14.9978094,E4 0.0,E5 0.0,E6 0.0}
DECL ATBg_Start_T AS_WDAT33={JobModeId -187662529,ParamSetId 687014726,StartTime 0.0,PreFlowTime 0.100000,Channel1 30.0000,Channel2 1.00000,Channel3 0.0,Channel4 0.0,Channel5 0.0,Channel6 0.0,Channel7 0.0,Channel8 0.0,PurgeTime 0.0}
DECL ATBg_Weld_T AW_WDAT33={JobModeId -187662529,ParamSetId -430485013,Velocity 0.00830000,Channel1 30.0000,Channel2 1.00000,Channel3 0.0,Channel4 0.0,Channel5 0.0,Channel6 0.0,Channel7 0.0,Channel8 0.0}
DECL WTCg_WeaveDefinition_T WV_WDAT33={Pattern #None,Length 4.00000,Amplitude 2.00000,Angle 0.0}
DECL FDAT FP61={TOOL_NO 1,BASE_NO 0,IPO_FRAME #BASE,POINT2[] " ",TQ_STATE FALSE}
DECL PDAT PPDAT47={ACC 100.000,APO_DIST 100.000,APO_MODE #CPTP,GEAR_JERK 50.0000}
DECL E6POS XP61={X 1395.70117,Y 144.395248,Z 1624.09387,A 63.4353790,B 85.7404404,C 145.440613,S 2,T 43,E1 15.0001278,E2 -131.762726,E3 14.9978094,E4 0.0,E5 0.0,E6 0.0}
DECL ATBg_Crater_T AC_WDAT34={JobModeId -187662529,ParamSetId -1375177600,CraterTime 0.100000,PostflowTime 0.100000,Channel1 30.0000,Channel2 1.00000,Channel3 0.0,Channel4 0.0,Channel5 0.0,Channel6 0.0,Channel7 0.0,Channel8 0.0,BurnBackTime 0.0}
DECL FDAT FP62={TOOL_NO 1,BASE_NO 0,IPO_FRAME #BASE,POINT2[] " ",TQ_STATE FALSE}
DECL LDAT LCPDAT16={ACC 100.000,APO_DIST 100.000,APO_FAC 50.0000,AXIS_VEL 100.000,AXIS_ACC 100.000,ORI_TYP #VAR,CIRC_TYP #BASE,JERK_FAC 50.0000,GEAR_JERK 50.0000,EXAX_IGN 0}
DECL E6POS XP62={X 1395.70117,Y 144.395248,Z 1624.09387,A 63.4353790,B 85.7404404,C 145.440613,S 2,T 43,E1 15.0001278,E2 -131.762726,E3 14.9978094,E4 0.0,E5 0.0,E6 0.0}
DECL E6POS XP63={X 1268.39099,Y 129.320740,Z 1747.43164,A 30.1052837,B 80.9914322,C 111.925606,S 2,T 43,E1 15.0001278,E2 -131.762726,E3 14.9978094,E4 0.0,E5 0.0,E6 0.0}
DECL FDAT FP63={TOOL_NO 1,BASE_NO 0,IPO_FRAME #BASE,POINT2[] " ",TQ_STATE FALSE}
DECL PDAT PPDAT48={VEL 100.000,ACC 100.000,APO_DIST 100.000,GEAR_JERK 50.0000,EXAX_IGN 3}
DECL E6POS XP64={X 1274.50281,Y -81.4749298,Z 1731.72900,A -48.8404579,B 83.1379852,C 41.7978439,S 2,T 10,E1 15.0001278,E2 -131.762726,E3 14.9978094,E4 0.0,E5 0.0,E6 0.0}
DECL FDAT FP64={TOOL_NO 1,BASE_NO 0,IPO_FRAME #BASE,POINT2[] " ",TQ_STATE FALSE}
DECL PDAT PPDAT49={VEL 100.000,ACC 100.000,APO_DIST 100.000,GEAR_JERK 50.0000,EXAX_IGN 3}
DECL E6POS XP65={X 1222.60547,Y 123.899391,Z 1786.00952,A 25.9520264,B 79.1208725,C 107.709618,S 2,T 43,E1 15.0001278,E2 -131.762726,E3 14.9978094,E4 0.0,E5 0.0,E6 0.0}
DECL FDAT FP65={TOOL_NO 1,BASE_NO 0,IPO_FRAME #BASE,POINT2[] " ",TQ_STATE FALSE}
DECL PDAT PPDAT50={VEL 100.000,ACC 100.000,APO_DIST 100.000,GEAR_JERK 50.0000,EXAX_IGN 3}
DECL PDAT PPDAT51={VEL 100.000,ACC 100.000,APO_DIST 100.000,GEAR_JERK 50.0000,EXAX_IGN 3}
ENDDAT
